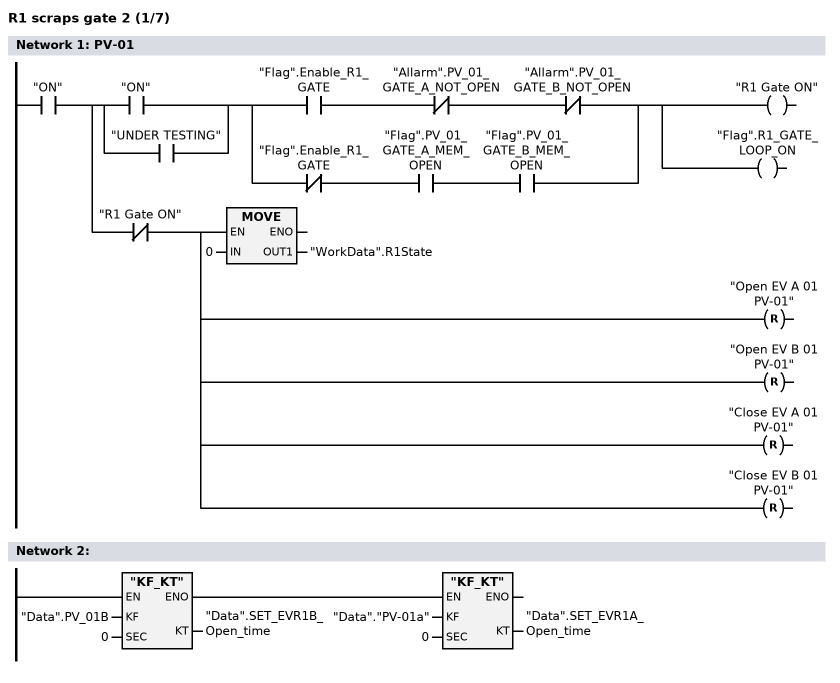
   RUNG wire#powerrail
      Contact( "ON" )
      wire#w1
      Contact( "ON" )
      wire#w2
      Contact( "Flag".Enable_R1_GATE )
      I_Contact( "Allarm".PV_01_GATE_A_NOT_OPEN )
      I_Contact( "Allarm".PV_01_GATE_B_NOT_OPEN )
      wire#w3
      Coil( "R1 Gate ON" )
   END_RUNG
   RUNG wire#w1
      Contact( "UNDER TESTING" )
   END_RUNG wire#w2
   RUNG wire#w2
      I_Contact( "Flag".Enable_R1_GATE )
      Contact( "Flag".PV_01_GATE_A_MEM_OPEN )
      Contact( "Flag".PV_01_GATE_B_MEM_OPEN )
   END_RUNG wire#w3
   RUNG wire#w3
      Coil( "Flag".R1_GATE_LOOP_ON )
   END_RUNG
   RUNG wire#w1
      I_Contact( "R1 Gate ON" )
      wire#w4
      { S7_GenerateENO := "TRUE" } Move(in := 0, out1 => "WorkData".R1State)
   END_RUNG
   RUNG wire#w4
      R_Coil( "Open EV A 01  PV-01" )
   END_RUNG
   RUNG wire#w4
      R_Coil( "Open EV B 01  PV-01" )
   END_RUNG
   RUNG wire#w4
      R_Coil( "Close EV A 01  PV-01" )
   END_RUNG
   RUNG wire#w4
      R_Coil( "Close EV B 01  PV-01" )
   END_RUNG
   // the same network as SCL:
   "R1 Gate ON" := "ON" AND ("ON" OR "UNDER TESTING") AND (("Flag".Enable_R1_GATE AND NOT "Allarm".PV_01_GATE_A_NOT_OPEN AND NOT "Allarm".PV_01_GATE_B_NOT_OPEN) OR (NOT "Flag".Enable_R1_GATE AND "Flag".PV_01_GATE_A_MEM_OPEN AND "Flag".PV_01_GATE_B_MEM_OPEN));
   "Flag".R1_GATE_LOOP_ON := "R1 Gate ON";
   IF "ON" AND NOT "R1 Gate ON" THEN
       "WorkData".R1State := 0;
       "Open EV A 01  PV-01" := FALSE;
       "Open EV B 01  PV-01" := FALSE;
       "Close EV A 01  PV-01" := FALSE;
       "Close EV B 01  PV-01" := FALSE;
   END_IF;
END_REGION

REGION Network 2
   RUNG wire#powerrail
      "KF_KT"(KF := "Data".PV_01B, SEC := 0, KT => "Data".SET_EVR1B_Open_time)
      "KF_KT"(KF := "Data"."PV-01a", SEC := 0, KT => "Data".SET_EVR1A_Open_time)
   END_RUNG
   // the same network as SCL:
   "KF_KT"(KF := "Data".PV_01B, SEC := 0, KT => "Data".SET_EVR1B_Open_time, ENO => #_w1);
   IF #_w1 THEN "KF_KT"(KF := "Data"."PV-01a", SEC := 0, KT => "Data".SET_EVR1A_Open_time); END_IF;
END_REGION

REGION Network 3: R1 gate loop PV-01
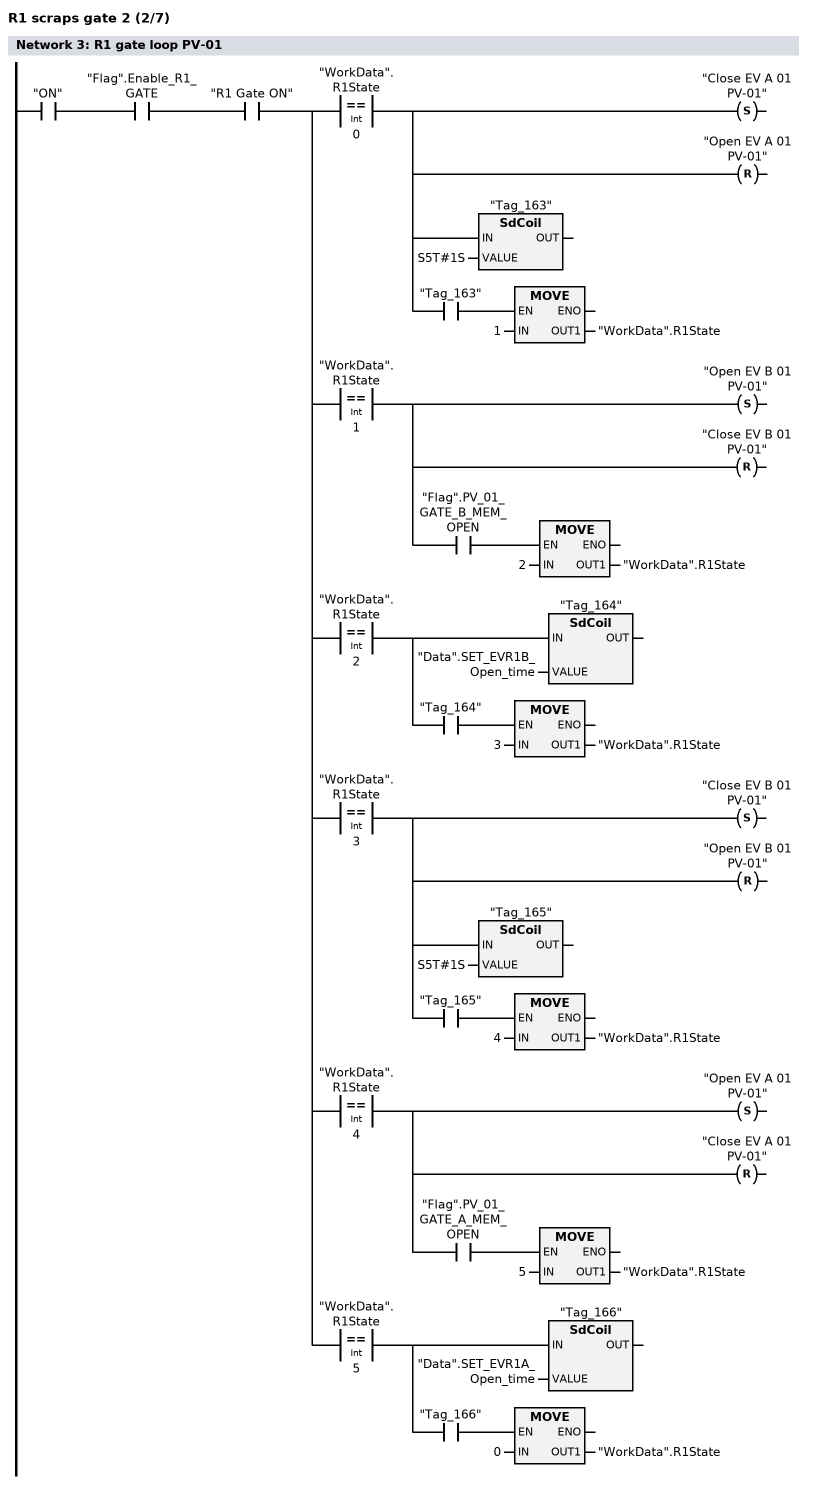
   // no SCL statement known for SdCoil: written as a call
   #_w1 := "ON" AND "Flag".Enable_R1_GATE AND "R1 Gate ON";
   #_w2 := #_w1 AND ("WorkData".R1State = 0);
   IF #_w2 THEN
       "Close EV A 01  PV-01" := TRUE;
       "Open EV A 01  PV-01" := FALSE;
   END_IF;
   SdCoil(in := #_w2, value := S5T#1S, operand := "Tag_163");
   IF #_w2 AND "Tag_163" THEN "WorkData".R1State := 1; END_IF;
   #_w3 := #_w1 AND ("WorkData".R1State = 1);
   IF #_w3 THEN
       "Open EV B 01  PV-01" := TRUE;
       "Close EV B 01  PV-01" := FALSE;
   END_IF;
   IF #_w3 AND "Flag".PV_01_GATE_B_MEM_OPEN THEN "WorkData".R1State := 2; END_IF;
   #_w4 := #_w1 AND ("WorkData".R1State = 2);
   SdCoil(in := #_w4, value := "Data".SET_EVR1B_Open_time, operand := "Tag_164");
   IF #_w4 AND "Tag_164" THEN "WorkData".R1State := 3; END_IF;
   #_w5 := #_w1 AND ("WorkData".R1State = 3);
   IF #_w5 THEN
       "Close EV B 01  PV-01" := TRUE;
       "Open EV B 01  PV-01" := FALSE;
   END_IF;
   SdCoil(in := #_w5, value := S5T#1S, operand := "Tag_165");
   IF #_w5 AND "Tag_165" THEN "WorkData".R1State := 4; END_IF;
   #_w6 := #_w1 AND ("WorkData".R1State = 4);
   IF #_w6 THEN
       "Open EV A 01  PV-01" := TRUE;
       "Close EV A 01  PV-01" := FALSE;
   END_IF;
   IF #_w6 AND "Flag".PV_01_GATE_A_MEM_OPEN THEN "WorkData".R1State := 5; END_IF;
   #_w7 := #_w1 AND ("WorkData".R1State = 5);
   SdCoil(in := #_w7, value := "Data".SET_EVR1A_Open_time, operand := "Tag_166");
   IF #_w7 AND "Tag_166" THEN "WorkData".R1State := 0; END_IF;
END_REGION

REGION Network 4: EVR4 scraps discharge door and Gates selector PV-01
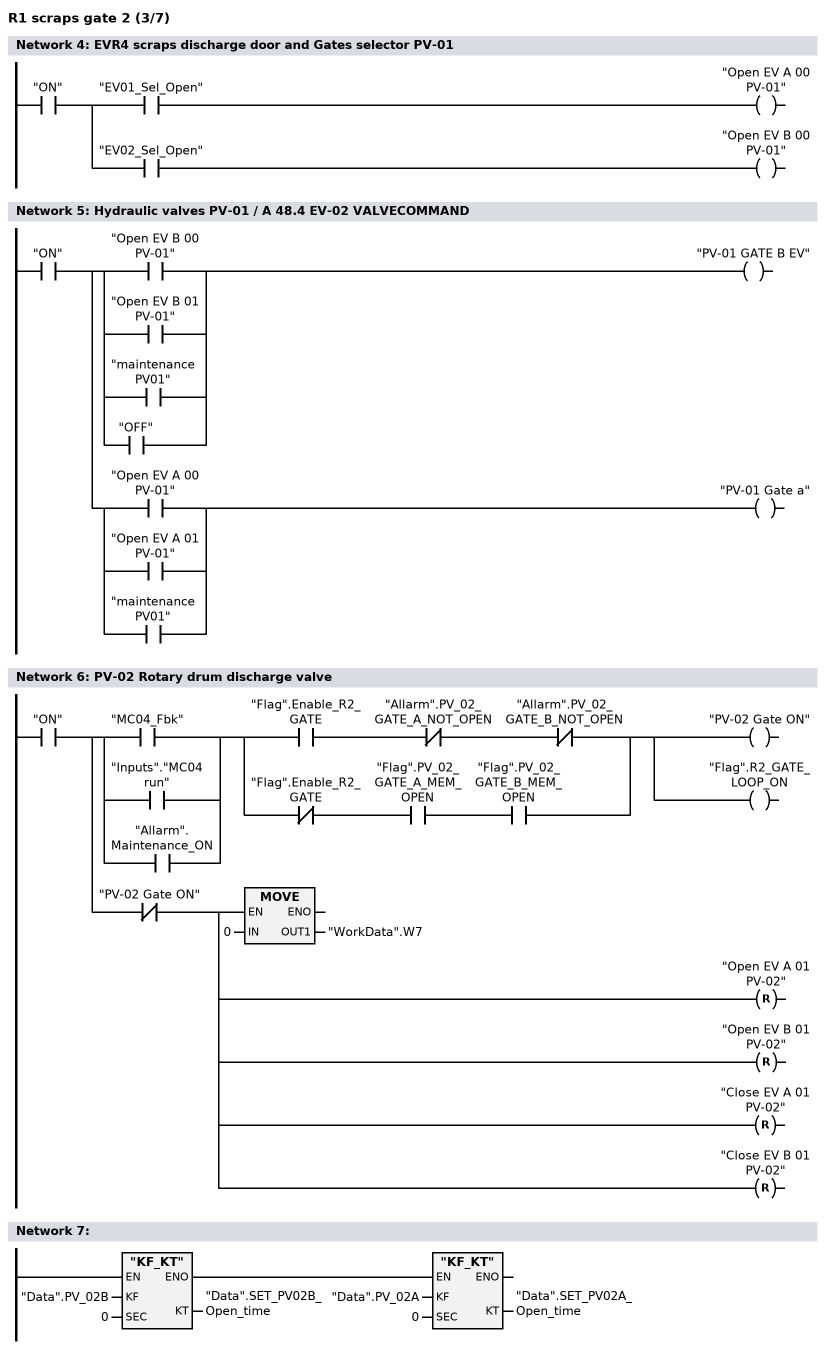
   RUNG wire#powerrail
      Contact( "ON" )
      wire#w1
      Contact( "EV01_Sel_Open" )
      Coil( "Open EV A 00 PV-01" )
   END_RUNG
   RUNG wire#w1
      Contact( "EV02_Sel_Open" )
      Coil( "Open EV B 00  PV-01" )
   END_RUNG
   // the same network as SCL:
   "Open EV A 00 PV-01" := "ON" AND "EV01_Sel_Open";
   "Open EV B 00  PV-01" := "ON" AND "EV02_Sel_Open";
END_REGION

REGION Network 5: Hydraulic valves PV-01 / A 48.4 EV-02 VALVECOMMAND
   RUNG wire#powerrail
      Contact( "ON" )
      wire#w1
      Contact( "Open EV B 00  PV-01" )
      wire#w2
      Coil( "PV-01 GATE B EV" )
   END_RUNG
   RUNG wire#w1
      Contact( "Open EV B 01  PV-01" )
   END_RUNG wire#w2
   RUNG wire#w1
      Contact( "maintenance PV01" )
   END_RUNG wire#w2
   RUNG wire#w1
      Contact( "OFF" )
   END_RUNG wire#w2
   RUNG wire#w1
      Contact( "Open EV A 00 PV-01" )
      wire#w3
      Coil( "PV-01 Gate a" )
   END_RUNG
   RUNG wire#w1
      Contact( "Open EV A 01  PV-01" )
   END_RUNG wire#w3
   RUNG wire#w1
      Contact( "maintenance PV01" )
   END_RUNG wire#w3
   // the same network as SCL:
   "PV-01 GATE B EV" := "ON" AND ("Open EV B 00  PV-01" OR "Open EV B 01  PV-01" OR "maintenance PV01" OR "OFF");
   "PV-01 Gate a" := "ON" AND ("Open EV A 00 PV-01" OR "Open EV A 01  PV-01" OR "maintenance PV01");
END_REGION

REGION Network 6: PV-02 Rotary drum discharge valve
   RUNG wire#powerrail
      Contact( "ON" )
      wire#w1
      Contact( "MC04_Fbk" )
      wire#w2
      Contact( "Flag".Enable_R2_GATE )
      I_Contact( "Allarm".PV_02_GATE_A_NOT_OPEN )
      I_Contact( "Allarm".PV_02_GATE_B_NOT_OPEN )
      wire#w3
      Coil( "PV-02 Gate ON" )
   END_RUNG
   RUNG wire#w1
      Contact( "Inputs"."MC04 run" )
   END_RUNG wire#w2
   RUNG wire#w1
      Contact( "Allarm".Maintenance_ON )
   END_RUNG wire#w2
   RUNG wire#w2
      I_Contact( "Flag".Enable_R2_GATE )
      Contact( "Flag".PV_02_GATE_A_MEM_OPEN )
      Contact( "Flag".PV_02_GATE_B_MEM_OPEN )
   END_RUNG wire#w3
   RUNG wire#w3
      Coil( "Flag".R2_GATE_LOOP_ON )
   END_RUNG
   RUNG wire#w1
      I_Contact( "PV-02 Gate ON" )
      wire#w4
      { S7_GenerateENO := "TRUE" } Move(in := 0, out1 => "WorkData".W7)
   END_RUNG
   RUNG wire#w4
      R_Coil( "Open EV A 01  PV-02" )
   END_RUNG
   RUNG wire#w4
      R_Coil( "Open EV B 01  PV-02" )
   END_RUNG
   RUNG wire#w4
      R_Coil( "Close EV A 01  PV-02" )
   END_RUNG
   RUNG wire#w4
      R_Coil( "Close EV B 01  PV-02" )
   END_RUNG
   // the same network as SCL:
   "PV-02 Gate ON" := "ON" AND ("MC04_Fbk" OR "Inputs"."MC04 run" OR "Allarm".Maintenance_ON) AND (("Flag".Enable_R2_GATE AND NOT "Allarm".PV_02_GATE_A_NOT_OPEN AND NOT "Allarm".PV_02_GATE_B_NOT_OPEN) OR (NOT "Flag".Enable_R2_GATE AND "Flag".PV_02_GATE_A_MEM_OPEN AND "Flag".PV_02_GATE_B_MEM_OPEN));
   "Flag".R2_GATE_LOOP_ON := "PV-02 Gate ON";
   IF "ON" AND NOT "PV-02 Gate ON" THEN
       "WorkData".W7 := 0;
       "Open EV A 01  PV-02" := FALSE;
       "Open EV B 01  PV-02" := FALSE;
       "Close EV A 01  PV-02" := FALSE;
       "Close EV B 01  PV-02" := FALSE;
   END_IF;
END_REGION

REGION Network 7
   RUNG wire#powerrail
      "KF_KT"(KF := "Data".PV_02B, SEC := 0, KT => "Data".SET_PV02B_Open_time)
      "KF_KT"(KF := "Data".PV_02A, SEC := 0, KT => "Data".SET_PV02A_Open_time)
   END_RUNG
   // the same network as SCL:
   "KF_KT"(KF := "Data".PV_02B, SEC := 0, KT => "Data".SET_PV02B_Open_time, ENO => #_w1);
   IF #_w1 THEN "KF_KT"(KF := "Data".PV_02A, SEC := 0, KT => "Data".SET_PV02A_Open_time); END_IF;
END_REGION

REGION Network 8: R1 gate loop PV-02
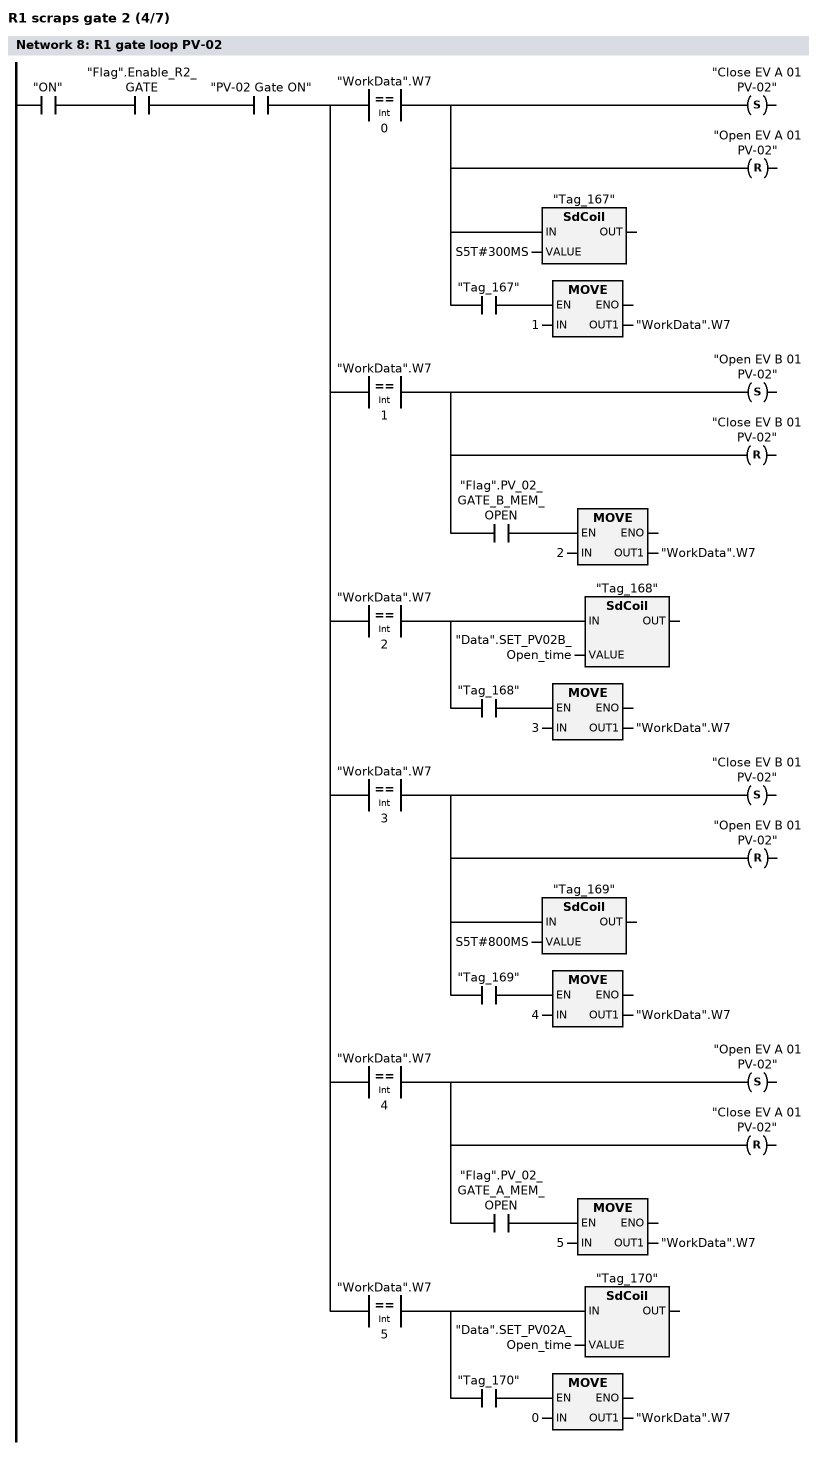
   // no SCL statement known for SdCoil: written as a call
   #_w1 := "ON" AND "Flag".Enable_R2_GATE AND "PV-02 Gate ON";
   #_w2 := #_w1 AND ("WorkData".W7 = 0);
   IF #_w2 THEN
       "Close EV A 01  PV-02" := TRUE;
       "Open EV A 01  PV-02" := FALSE;
   END_IF;
   SdCoil(in := #_w2, value := S5T#300MS, operand := "Tag_167");
   IF #_w2 AND "Tag_167" THEN "WorkData".W7 := 1; END_IF;
   #_w3 := #_w1 AND ("WorkData".W7 = 1);
   IF #_w3 THEN
       "Open EV B 01  PV-02" := TRUE;
       "Close EV B 01  PV-02" := FALSE;
   END_IF;
   IF #_w3 AND "Flag".PV_02_GATE_B_MEM_OPEN THEN "WorkData".W7 := 2; END_IF;
   #_w4 := #_w1 AND ("WorkData".W7 = 2);
   SdCoil(in := #_w4, value := "Data".SET_PV02B_Open_time, operand := "Tag_168");
   IF #_w4 AND "Tag_168" THEN "WorkData".W7 := 3; END_IF;
   #_w5 := #_w1 AND ("WorkData".W7 = 3);
   IF #_w5 THEN
       "Close EV B 01  PV-02" := TRUE;
       "Open EV B 01  PV-02" := FALSE;
   END_IF;
   SdCoil(in := #_w5, value := S5T#800MS, operand := "Tag_169");
   IF #_w5 AND "Tag_169" THEN "WorkData".W7 := 4; END_IF;
   #_w6 := #_w1 AND ("WorkData".W7 = 4);
   IF #_w6 THEN
       "Open EV A 01  PV-02" := TRUE;
       "Close EV A 01  PV-02" := FALSE;
   END_IF;
   IF #_w6 AND "Flag".PV_02_GATE_A_MEM_OPEN THEN "WorkData".W7 := 5; END_IF;
   #_w7 := #_w1 AND ("WorkData".W7 = 5);
   SdCoil(in := #_w7, value := "Data".SET_PV02A_Open_time, operand := "Tag_170");
   IF #_w7 AND "Tag_170" THEN "WorkData".W7 := 0; END_IF;
END_REGION

REGION Network 9: EVR4 scraps discharge door and Gates selector PV-02
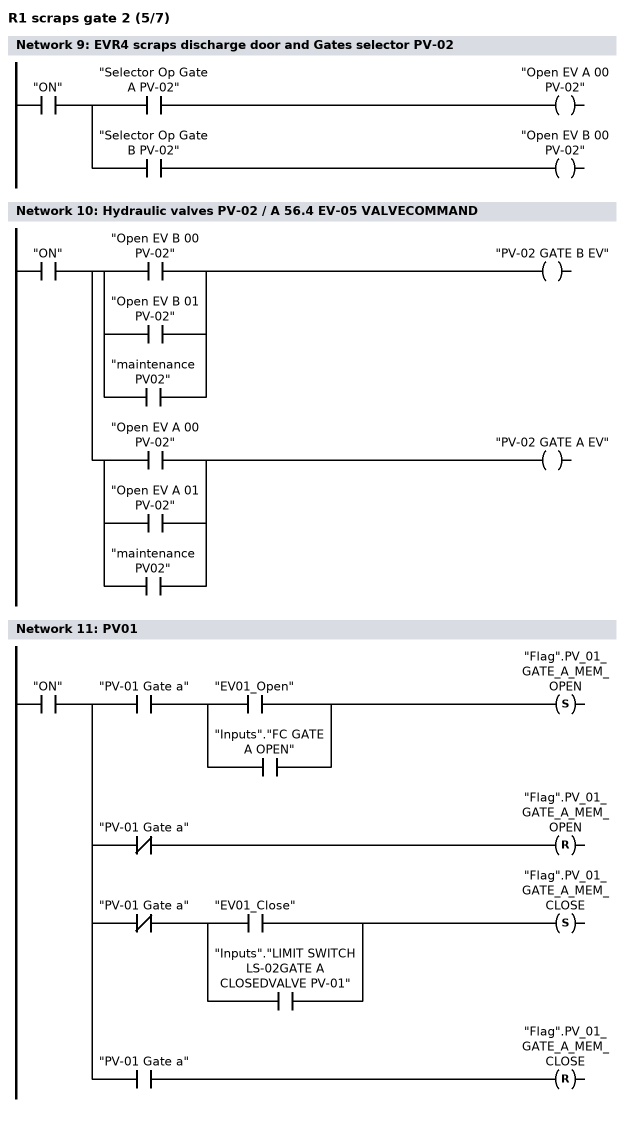
   RUNG wire#powerrail
      Contact( "ON" )
      wire#w1
      Contact( "Selector Op Gate A PV-02" )
      Coil( "Open EV A 00 PV-02" )
   END_RUNG
   RUNG wire#w1
      Contact( "Selector Op Gate B PV-02" )
      Coil( "Open EV B 00  PV-02" )
   END_RUNG
   // the same network as SCL:
   "Open EV A 00 PV-02" := "ON" AND "Selector Op Gate A PV-02";
   "Open EV B 00  PV-02" := "ON" AND "Selector Op Gate B PV-02";
END_REGION

REGION Network 10: Hydraulic valves PV-02 / A 56.4 EV-05 VALVECOMMAND
   RUNG wire#powerrail
      Contact( "ON" )
      wire#w1
      Contact( "Open EV B 00  PV-02" )
      wire#w2
      Coil( "PV-02 GATE B EV" )
   END_RUNG
   RUNG wire#w1
      Contact( "Open EV B 01  PV-02" )
   END_RUNG wire#w2
   RUNG wire#w1
      Contact( "maintenance PV02" )
   END_RUNG wire#w2
   RUNG wire#w1
      Contact( "Open EV A 00 PV-02" )
      wire#w3
      Coil( "PV-02 GATE A EV" )
   END_RUNG
   RUNG wire#w1
      Contact( "Open EV A 01  PV-02" )
   END_RUNG wire#w3
   RUNG wire#w1
      Contact( "maintenance PV02" )
   END_RUNG wire#w3
   // the same network as SCL:
   "PV-02 GATE B EV" := "ON" AND ("Open EV B 00  PV-02" OR "Open EV B 01  PV-02" OR "maintenance PV02");
   "PV-02 GATE A EV" := "ON" AND ("Open EV A 00 PV-02" OR "Open EV A 01  PV-02" OR "maintenance PV02");
END_REGION

REGION Network 11: PV01
   RUNG wire#powerrail
      Contact( "ON" )
      wire#w1
      Contact( "PV-01 Gate a" )
      wire#w2
      Contact( "EV01_Open" )
      wire#w3
      S_Coil( "Flag".PV_01_GATE_A_MEM_OPEN )
   END_RUNG
   RUNG wire#w2
      Contact( "Inputs"."FC GATE A OPEN" )
   END_RUNG wire#w3
   RUNG wire#w1
      I_Contact( "PV-01 Gate a" )
      R_Coil( "Flag".PV_01_GATE_A_MEM_OPEN )
   END_RUNG
   RUNG wire#w1
      I_Contact( "PV-01 Gate a" )
      wire#w4
      Contact( "EV01_Close" )
      wire#w5
      S_Coil( "Flag".PV_01_GATE_A_MEM_CLOSE )
   END_RUNG
   RUNG wire#w4
      Contact( "Inputs"."LIMIT SWITCH LS-02GATE A CLOSEDVALVE PV-01" )
   END_RUNG wire#w5
   RUNG wire#w1
      Contact( "PV-01 Gate a" )
      R_Coil( "Flag".PV_01_GATE_A_MEM_CLOSE )
   END_RUNG
   // the same network as SCL:
   IF "ON" AND "PV-01 Gate a" AND ("EV01_Open" OR "Inputs"."FC GATE A OPEN") THEN
       "Flag".PV_01_GATE_A_MEM_OPEN := TRUE;
   END_IF;
   IF "ON" AND NOT "PV-01 Gate a" THEN "Flag".PV_01_GATE_A_MEM_OPEN := FALSE; END_IF;
   IF "ON" AND NOT "PV-01 Gate a" AND ("EV01_Close" OR "Inputs"."LIMIT SWITCH LS-02GATE A CLOSEDVALVE PV-01") THEN
       "Flag".PV_01_GATE_A_MEM_CLOSE := TRUE;
   END_IF;
   IF "ON" AND "PV-01 Gate a" THEN "Flag".PV_01_GATE_A_MEM_CLOSE := FALSE; END_IF;
END_REGION

REGION Network 12: PV01
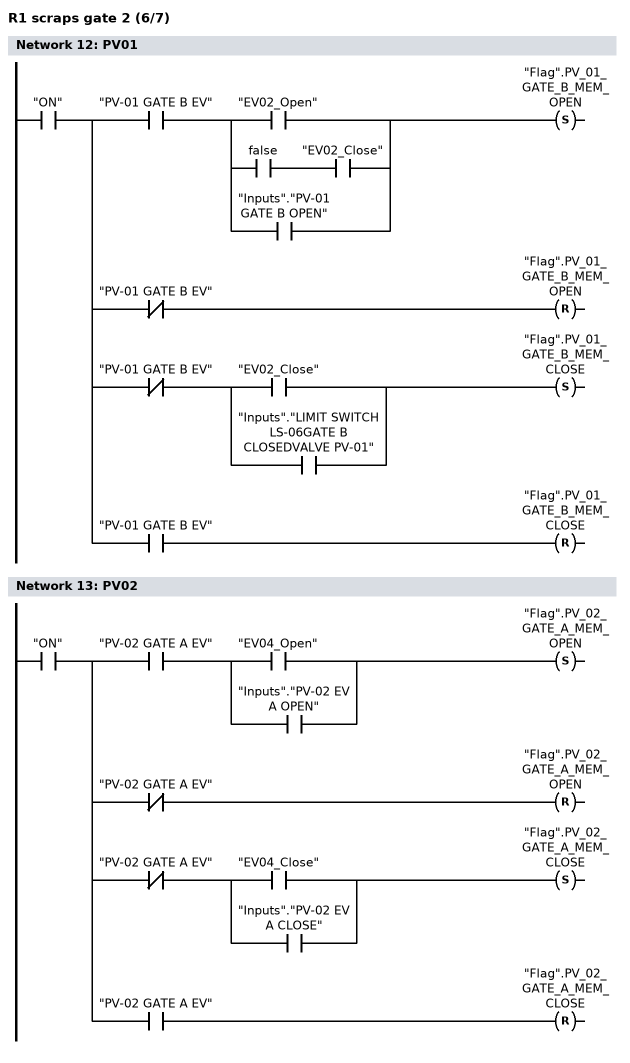
   RUNG wire#powerrail
      Contact( "ON" )
      wire#w1
      Contact( "PV-01 GATE B EV" )
      wire#w2
      Contact( "EV02_Open" )
      wire#w3
      S_Coil( "Flag".PV_01_GATE_B_MEM_OPEN )
   END_RUNG
   RUNG wire#w2
      Contact( false )
      Contact( "EV02_Close" )
   END_RUNG wire#w3
   RUNG wire#w2
      Contact( "Inputs"."PV-01 GATE B OPEN" )
   END_RUNG wire#w3
   RUNG wire#w1
      I_Contact( "PV-01 GATE B EV" )
      R_Coil( "Flag".PV_01_GATE_B_MEM_OPEN )
   END_RUNG
   RUNG wire#w1
      I_Contact( "PV-01 GATE B EV" )
      wire#w4
      Contact( "EV02_Close" )
      wire#w5
      S_Coil( "Flag".PV_01_GATE_B_MEM_CLOSE )
   END_RUNG
   RUNG wire#w4
      Contact( "Inputs"."LIMIT SWITCH LS-06GATE B CLOSEDVALVE PV-01" )
   END_RUNG wire#w5
   RUNG wire#w1
      Contact( "PV-01 GATE B EV" )
      R_Coil( "Flag".PV_01_GATE_B_MEM_CLOSE )
   END_RUNG
   // the same network as SCL:
   IF "ON" AND "PV-01 GATE B EV" AND ("EV02_Open" OR (false AND "EV02_Close") OR "Inputs"."PV-01 GATE B OPEN") THEN
       "Flag".PV_01_GATE_B_MEM_OPEN := TRUE;
   END_IF;
   IF "ON" AND NOT "PV-01 GATE B EV" THEN "Flag".PV_01_GATE_B_MEM_OPEN := FALSE; END_IF;
   IF "ON" AND NOT "PV-01 GATE B EV" AND ("EV02_Close" OR "Inputs"."LIMIT SWITCH LS-06GATE B CLOSEDVALVE PV-01") THEN
       "Flag".PV_01_GATE_B_MEM_CLOSE := TRUE;
   END_IF;
   IF "ON" AND "PV-01 GATE B EV" THEN "Flag".PV_01_GATE_B_MEM_CLOSE := FALSE; END_IF;
END_REGION

REGION Network 13: PV02
   RUNG wire#powerrail
      Contact( "ON" )
      wire#w1
      Contact( "PV-02 GATE A EV" )
      wire#w2
      Contact( "EV04_Open" )
      wire#w3
      S_Coil( "Flag".PV_02_GATE_A_MEM_OPEN )
   END_RUNG
   RUNG wire#w2
      Contact( "Inputs"."PV-02 EV A OPEN" )
   END_RUNG wire#w3
   RUNG wire#w1
      I_Contact( "PV-02 GATE A EV" )
      R_Coil( "Flag".PV_02_GATE_A_MEM_OPEN )
   END_RUNG
   RUNG wire#w1
      I_Contact( "PV-02 GATE A EV" )
      wire#w4
      Contact( "EV04_Close" )
      wire#w5
      S_Coil( "Flag".PV_02_GATE_A_MEM_CLOSE )
   END_RUNG
   RUNG wire#w4
      Contact( "Inputs"."PV-02 EV A CLOSE" )
   END_RUNG wire#w5
   RUNG wire#w1
      Contact( "PV-02 GATE A EV" )
      R_Coil( "Flag".PV_02_GATE_A_MEM_CLOSE )
   END_RUNG
   // the same network as SCL:
   IF "ON" AND "PV-02 GATE A EV" AND ("EV04_Open" OR "Inputs"."PV-02 EV A OPEN") THEN
       "Flag".PV_02_GATE_A_MEM_OPEN := TRUE;
   END_IF;
   IF "ON" AND NOT "PV-02 GATE A EV" THEN "Flag".PV_02_GATE_A_MEM_OPEN := FALSE; END_IF;
   IF "ON" AND NOT "PV-02 GATE A EV" AND ("EV04_Close" OR "Inputs"."PV-02 EV A CLOSE") THEN
       "Flag".PV_02_GATE_A_MEM_CLOSE := TRUE;
   END_IF;
   IF "ON" AND "PV-02 GATE A EV" THEN "Flag".PV_02_GATE_A_MEM_CLOSE := FALSE; END_IF;
END_REGION

REGION Network 14: PV02
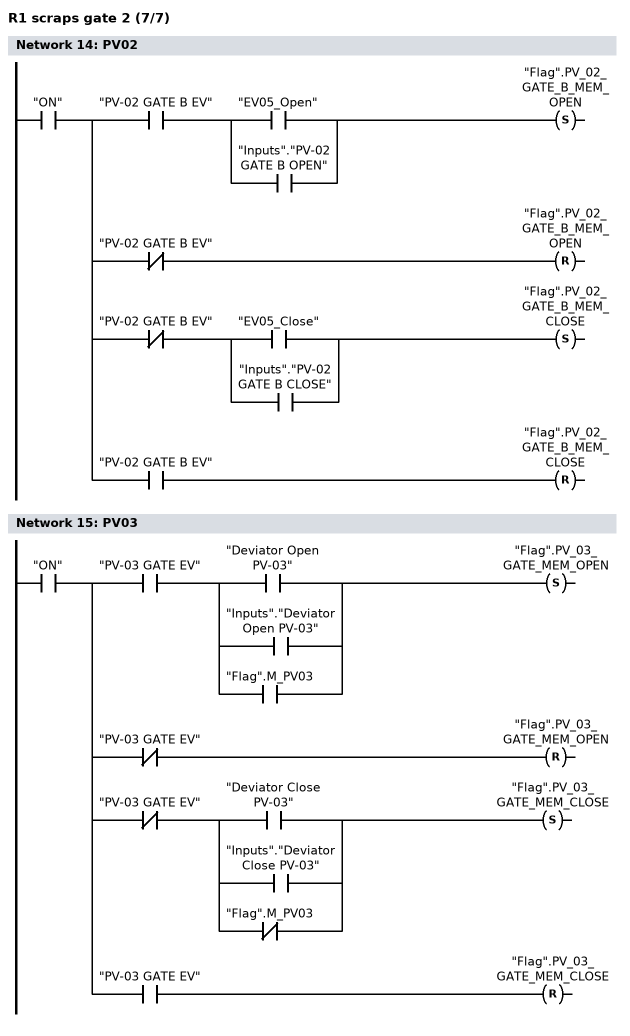
   RUNG wire#powerrail
      Contact( "ON" )
      wire#w1
      Contact( "PV-02 GATE B EV" )
      wire#w2
      Contact( "EV05_Open" )
      wire#w3
      S_Coil( "Flag".PV_02_GATE_B_MEM_OPEN )
   END_RUNG
   RUNG wire#w2
      Contact( "Inputs"."PV-02 GATE B OPEN" )
   END_RUNG wire#w3
   RUNG wire#w1
      I_Contact( "PV-02 GATE B EV" )
      R_Coil( "Flag".PV_02_GATE_B_MEM_OPEN )
   END_RUNG
   RUNG wire#w1
      I_Contact( "PV-02 GATE B EV" )
      wire#w4
      Contact( "EV05_Close" )
      wire#w5
      S_Coil( "Flag".PV_02_GATE_B_MEM_CLOSE )
   END_RUNG
   RUNG wire#w4
      Contact( "Inputs"."PV-02 GATE B CLOSE" )
   END_RUNG wire#w5
   RUNG wire#w1
      Contact( "PV-02 GATE B EV" )
      R_Coil( "Flag".PV_02_GATE_B_MEM_CLOSE )
   END_RUNG
   // the same network as SCL:
   IF "ON" AND "PV-02 GATE B EV" AND ("EV05_Open" OR "Inputs"."PV-02 GATE B OPEN") THEN
       "Flag".PV_02_GATE_B_MEM_OPEN := TRUE;
   END_IF;
   IF "ON" AND NOT "PV-02 GATE B EV" THEN "Flag".PV_02_GATE_B_MEM_OPEN := FALSE; END_IF;
   IF "ON" AND NOT "PV-02 GATE B EV" AND ("EV05_Close" OR "Inputs"."PV-02 GATE B CLOSE") THEN
       "Flag".PV_02_GATE_B_MEM_CLOSE := TRUE;
   END_IF;
   IF "ON" AND "PV-02 GATE B EV" THEN "Flag".PV_02_GATE_B_MEM_CLOSE := FALSE; END_IF;
END_REGION

REGION Network 15: PV03
   RUNG wire#powerrail
      Contact( "ON" )
      wire#w1
      Contact( "PV-03 GATE EV" )
      wire#w2
      Contact( "Deviator Open PV-03" )
      wire#w3
      S_Coil( "Flag".PV_03_GATE_MEM_OPEN )
   END_RUNG
   RUNG wire#w2
      Contact( "Inputs"."Deviator Open PV-03" )
   END_RUNG wire#w3
   RUNG wire#w2
      Contact( "Flag".M_PV03 )
   END_RUNG wire#w3
   RUNG wire#w1
      I_Contact( "PV-03 GATE EV" )
      R_Coil( "Flag".PV_03_GATE_MEM_OPEN )
   END_RUNG
   RUNG wire#w1
      I_Contact( "PV-03 GATE EV" )
      wire#w4
      Contact( "Deviator Close PV-03" )
      wire#w5
      S_Coil( "Flag".PV_03_GATE_MEM_CLOSE )
   END_RUNG
   RUNG wire#w4
      Contact( "Inputs"."Deviator Close PV-03" )
   END_RUNG wire#w5
   RUNG wire#w4
      I_Contact( "Flag".M_PV03 )
   END_RUNG wire#w5
   RUNG wire#w1
      Contact( "PV-03 GATE EV" )
      R_Coil( "Flag".PV_03_GATE_MEM_CLOSE )
   END_RUNG
   // the same network as SCL:
   IF "ON" AND "PV-03 GATE EV" AND ("Deviator Open PV-03" OR "Inputs"."Deviator Open PV-03" OR "Flag".M_PV03) THEN
       "Flag".PV_03_GATE_MEM_OPEN := TRUE;
   END_IF;
   IF "ON" AND NOT "PV-03 GATE EV" THEN "Flag".PV_03_GATE_MEM_OPEN := FALSE; END_IF;
   IF "ON" AND NOT "PV-03 GATE EV" AND ("Deviator Close PV-03" OR "Inputs"."Deviator Close PV-03" OR NOT "Flag".M_PV03) THEN
       "Flag".PV_03_GATE_MEM_CLOSE := TRUE;
   END_IF;
   IF "ON" AND "PV-03 GATE EV" THEN "Flag".PV_03_GATE_MEM_CLOSE := FALSE; END_IF;
END_REGION
END_FUNCTION

FUNCTION "KF_KT" : Void   // FC109, STL
TITLE = Conversione tempo KF => KT - Max. 9990 secondi / Converion time KF=>KT - Max. 9990 seconds
{ S7_Optimized_Access := 'FALSE' }
VERSION : 0.1
   VAR_INPUT
      KF : Int;   // Secondi o decimi / Seconds or tenths
      SEC : Bool;   // TRUE = secondi, FALSE = decimi / TRUE = seconds, FALSE = tenths
   END_VAR
   VAR_OUTPUT
      KT : Word;
   END_VAR
BEGIN

REGION Network 1
   // Converte il valore di tempo KF espresso in secondi o in decimi di secondo nel 
   // corrispondente preset in formato S5T (KT); in SEC occorre specificare TRUE se
   // il valore di partenza è espresso in secondi, FALSE se in decimi.
   // Converts the KF time value expressed in seconds or tenths of a second to 
   // corresponding preset in S5T (KT) format; in SEC you must specify TRUE if
   // the starting value is expressed in seconds, FALSE if in tenths

         L     0;
         T     #KT;
         L     #KF;  // tempo in secondi o decimi
         >=I;
         BEC;  // esci se <= 0

         AN    #SEC;
         JC    X1;  // se secondi
         L     10;  // x 10
         *I;  // Tempo in decimi

   // Tra 0 e 9.9 secondi
   X1:   L     99;
         >D;
         JC    X2;
         TAK;  // Tempo in decimi
         ITB;  // Converti in BCD
         SLW   4;  // aggiungi uno zero a destra (x10)
         JU    ESC;  // Base 0 = decine di ms

   // Tra 10.0 e 99.9 secondi
   X2:   TAK;  // Tempo in decimi
         L     999;
         >D;
         JC    X3;
         TAK;  // Tempo in decimi
         ITB;  // Converti in BCD
         L     16#1000;  // Base 1 = decimi
         JU    OR;

   // Tra 100.0 e 999.9 secondi
   X3:   TAK;  // Tempo in decimi
         +     5;  // +5 per arrotondamento
         L     9999;
         >D;
         JC    X4;
         TAK;  // Tempo in decimi
         DTB;  // converti in BCD
         SRD   4;  // Sposta a destra di 1 cifra (/10)
         L     16#2000;  // Base 2 = secondi
         JU    OR;

   // Tra 1000.0 e 9990.0 secondi
   X4:   TAK;  // Tempo in decimi
         +     45;  // +50 (45+5) per arrotondamento
         L     99900;
         >D;
         JC    X5;
         TAK;  // Tempo in decimi
         DTB;  // converti in BCD
         SRD   8;  // Sposta a destra di 2 cifre (/100)
         L     16#3000;  // Base 3 = decine di secondi
         JU    OR;

   // Oltre 9990.0 secondi
   X5:   L     16#3999;  // Massimo tempo possibile
         JU    ESC;

   // Uscita
   OR:   OW;  // Aggiungi la base
   ESC:  T     #KT;  // Uscita
END_REGION
END_FUNCTION

ORGANIZATION_BLOCK "Main"   // OB1, LAD, ProgramCycle
TITLE = Main program
{ S7_Optimized_Access := 'FALSE' }
VERSION : 0.1
   VAR_TEMP
      TodayDate : Date;
      ReadClkRetValue : Int;
      TodayDateTime : Date_And_Time;
      spare : DWord;
      spare_1 : DWord;
      spare_2 : DWord;
   END_VAR
   VAR_TEMP   // added for the SCL form of the ladder/FBD networks
      _w1 : Bool;
      _w2 : Bool;
      _w3 : Bool;
   END_VAR
BEGIN

REGION Network 1: SIMULATION
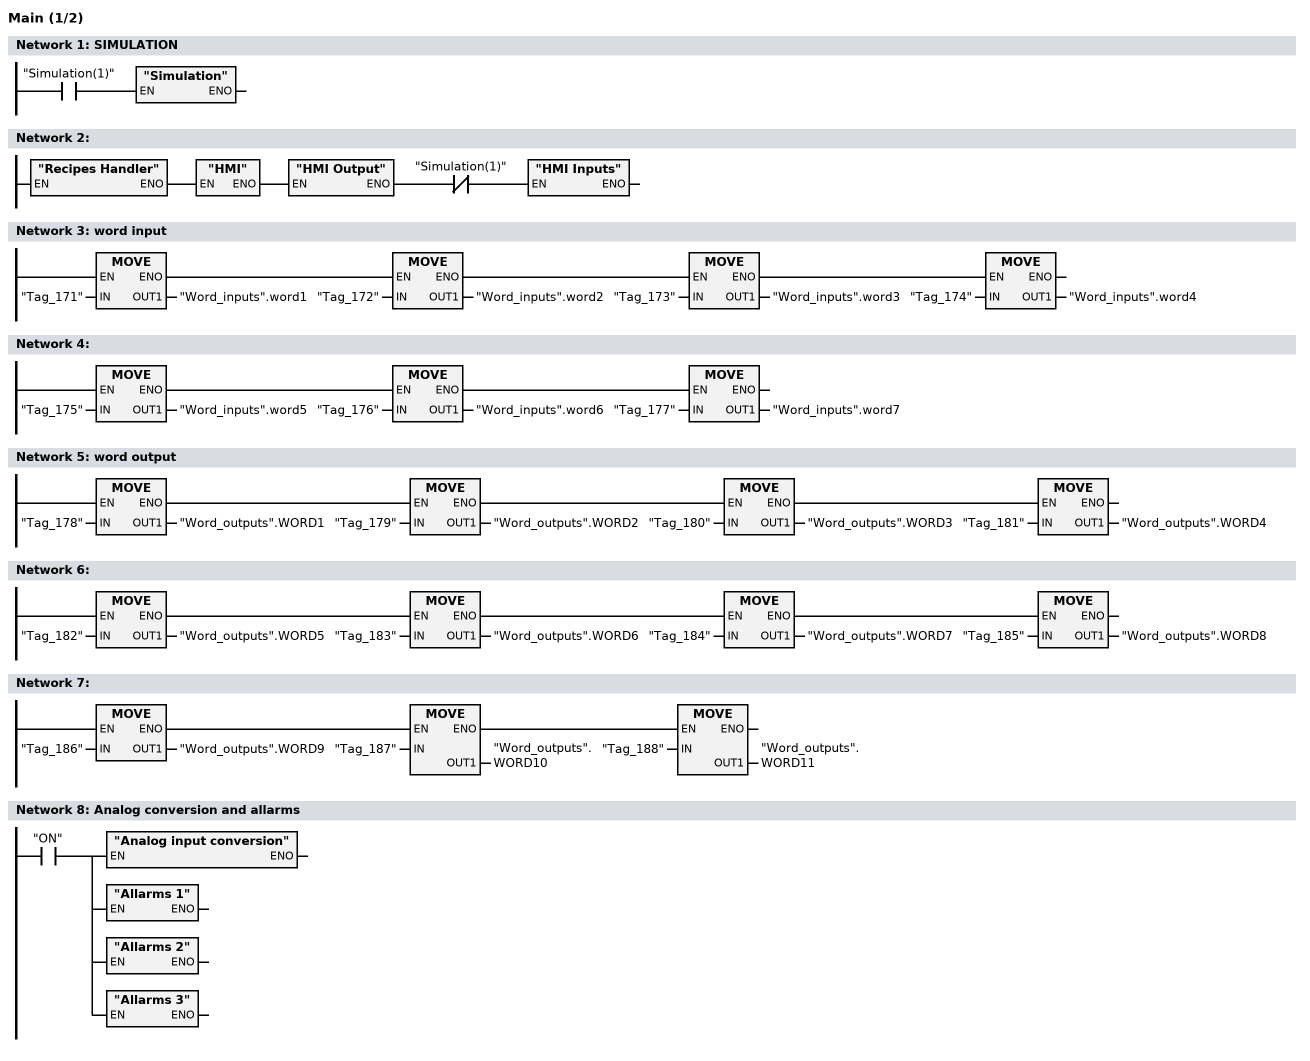
   RUNG wire#powerrail
      Contact( "Simulation(1)" )
      "Simulation"()
   END_RUNG
   // the same network as SCL:
   IF "Simulation(1)" THEN "Simulation"(); END_IF;
END_REGION

REGION Network 2
   RUNG wire#powerrail
      "Recipes Handler"()
      "HMI"()
      "HMI Output"()
      I_Contact( "Simulation(1)" )
      "HMI Inputs"()
   END_RUNG
   // the same network as SCL:
   "Recipes Handler"(ENO => #_w1);
   "HMI"(EN := #_w1, ENO => #_w2);
   "HMI Output"(EN := #_w2, ENO => #_w3);
   IF #_w3 AND NOT "Simulation(1)" THEN "HMI Inputs"(); END_IF;
END_REGION

REGION Network 3: word input
   RUNG wire#powerrail
      { S7_GenerateENO := "TRUE" } Move(in := "Tag_171", out1 => "Word_inputs".word1)
      { S7_GenerateENO := "TRUE" } Move(in := "Tag_172", out1 => "Word_inputs".word2)
      { S7_GenerateENO := "TRUE" } Move(in := "Tag_173", out1 => "Word_inputs".word3)
      { S7_GenerateENO := "TRUE" } Move(in := "Tag_174", out1 => "Word_inputs".word4)
   END_RUNG
   // the same network as SCL:
   // ENO of a box is taken as its EN; it also drops when the box reports an error
   "Word_inputs".word1 := "Tag_171";
   "Word_inputs".word2 := "Tag_172";
   "Word_inputs".word3 := "Tag_173";
   "Word_inputs".word4 := "Tag_174";
END_REGION

REGION Network 4
   RUNG wire#powerrail
      { S7_GenerateENO := "TRUE" } Move(in := "Tag_175", out1 => "Word_inputs".word5)
      { S7_GenerateENO := "TRUE" } Move(in := "Tag_176", out1 => "Word_inputs".word6)
      { S7_GenerateENO := "TRUE" } Move(in := "Tag_177", out1 => "Word_inputs".word7)
   END_RUNG
   // the same network as SCL:
   // ENO of a box is taken as its EN; it also drops when the box reports an error
   "Word_inputs".word5 := "Tag_175";
   "Word_inputs".word6 := "Tag_176";
   "Word_inputs".word7 := "Tag_177";
END_REGION

REGION Network 5: word output
   RUNG wire#powerrail
      { S7_GenerateENO := "TRUE" } Move(in := "Tag_178", out1 => "Word_outputs".WORD1)
      { S7_GenerateENO := "TRUE" } Move(in := "Tag_179", out1 => "Word_outputs".WORD2)
      { S7_GenerateENO := "TRUE" } Move(in := "Tag_180", out1 => "Word_outputs".WORD3)
      { S7_GenerateENO := "TRUE" } Move(in := "Tag_181", out1 => "Word_outputs".WORD4)
   END_RUNG
   // the same network as SCL:
   // ENO of a box is taken as its EN; it also drops when the box reports an error
   "Word_outputs".WORD1 := "Tag_178";
   "Word_outputs".WORD2 := "Tag_179";
   "Word_outputs".WORD3 := "Tag_180";
   "Word_outputs".WORD4 := "Tag_181";
END_REGION

REGION Network 6
   RUNG wire#powerrail
      { S7_GenerateENO := "TRUE" } Move(in := "Tag_182", out1 => "Word_outputs".WORD5)
      { S7_GenerateENO := "TRUE" } Move(in := "Tag_183", out1 => "Word_outputs".WORD6)
      { S7_GenerateENO := "TRUE" } Move(in := "Tag_184", out1 => "Word_outputs".WORD7)
      { S7_GenerateENO := "TRUE" } Move(in := "Tag_185", out1 => "Word_outputs".WORD8)
   END_RUNG
   // the same network as SCL:
   // ENO of a box is taken as its EN; it also drops when the box reports an error
   "Word_outputs".WORD5 := "Tag_182";
   "Word_outputs".WORD6 := "Tag_183";
   "Word_outputs".WORD7 := "Tag_184";
   "Word_outputs".WORD8 := "Tag_185";
END_REGION

REGION Network 7
   RUNG wire#powerrail
      { S7_GenerateENO := "TRUE" } Move(in := "Tag_186", out1 => "Word_outputs".WORD9)
      { S7_GenerateENO := "TRUE" } Move(in := "Tag_187", out1 => "Word_outputs".WORD10)
      { S7_GenerateENO := "TRUE" } Move(in := "Tag_188", out1 => "Word_outputs".WORD11)
   END_RUNG
   // the same network as SCL:
   // ENO of a box is taken as its EN; it also drops when the box reports an error
   "Word_outputs".WORD9 := "Tag_186";
   "Word_outputs".WORD10 := "Tag_187";
   "Word_outputs".WORD11 := "Tag_188";
END_REGION

REGION Network 8: Analog conversion and allarms
   RUNG wire#powerrail
      Contact( "ON" )
      wire#w1
      "Analog input conversion"()
   END_RUNG
   RUNG wire#w1
      "Allarms 1"()
   END_RUNG
   RUNG wire#w1
      "Allarms 2"()
   END_RUNG
   RUNG wire#w1
      "Allarms 3"()
   END_RUNG
   // the same network as SCL:
   #_w1 := "ON";
   IF #_w1 THEN
       "Analog input conversion"();
       "Allarms 1"();
       "Allarms 2"();
       "Allarms 3"();
   END_IF;
END_REGION

REGION Network 9: Motors valve and burner
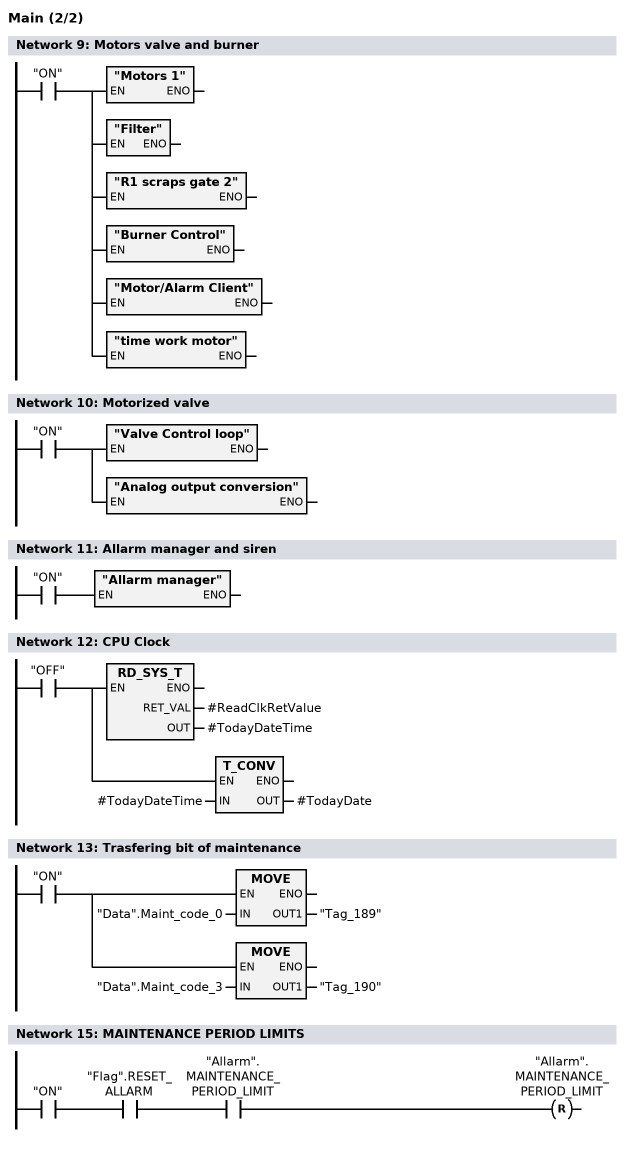
   RUNG wire#powerrail
      Contact( "ON" )
      wire#w1
      "Motors 1"()
   END_RUNG
   RUNG wire#w1
      "Filter"()
   END_RUNG
   RUNG wire#w1
      "R1 scraps gate 2"()
   END_RUNG
   RUNG wire#w1
      "Burner Control"()
   END_RUNG
   RUNG wire#w1
      "Motor/Alarm Client"()
   END_RUNG
   RUNG wire#w1
      "time work motor"()
   END_RUNG
   // the same network as SCL:
   #_w1 := "ON";
   IF #_w1 THEN
       "Motors 1"();
       "Filter"();
       "R1 scraps gate 2"();
       "Burner Control"();
       "Motor/Alarm Client"();
       "time work motor"();
   END_IF;
END_REGION

REGION Network 10: Motorized valve
   RUNG wire#powerrail
      Contact( "ON" )
      wire#w1
      "Valve Control loop"()
   END_RUNG
   RUNG wire#w1
      "Analog output conversion"()
   END_RUNG
   // the same network as SCL:
   #_w1 := "ON";
   IF #_w1 THEN
       "Valve Control loop"();
       "Analog output conversion"();
   END_IF;
END_REGION

REGION Network 11: Allarm manager and siren
   RUNG wire#powerrail
      Contact( "ON" )
      "Allarm manager"()
   END_RUNG
   // the same network as SCL:
   IF "ON" THEN "Allarm manager"(); END_IF;
END_REGION

REGION Network 12: CPU Clock
   #_w1 := "OFF";
   IF #_w1 THEN
       #ReadClkRetValue := RD_SYS_T(OUT => #TodayDateTime);
       #TodayDate := T_CONV(IN := #TodayDateTime);
   END_IF;
END_REGION

REGION Network 13: Trasfering bit of maintenance
   RUNG wire#powerrail
      Contact( "ON" )
      wire#w1
      { S7_GenerateENO := "TRUE" } Move(in := "Data".Maint_code_0, out1 => "Tag_189")
   END_RUNG
   RUNG wire#w1
      { S7_GenerateENO := "TRUE" } Move(in := "Data".Maint_code_3, out1 => "Tag_190")
   END_RUNG
   // the same network as SCL:
   IF "ON" THEN
       "Tag_189" := "Data".Maint_code_0;
       "Tag_190" := "Data".Maint_code_3;
   END_IF;
END_REGION

REGION Network 14 (STL): MAINTENANCE PERIOD LIMITS
         L     "Data".Maint_code_1;

         L     16972;
         ==I;
         JC    M001;

         CALL  RD_SYS_T
         ( RET_VAL := #ReadClkRetValue,
           OUT     := #TodayDateTime
         );

         CALL  T_CONV
         ( IN  := #TodayDateTime,
           OUT := #TodayDate
         );

         L     #TodayDate;
         L     D#2026-01-01;


         >=I;
         S     "Allarm".MAINTENANCE_PERIOD_LIMIT;

   M001: NOP   0;
END_REGION

REGION Network 15: MAINTENANCE PERIOD LIMITS
   RUNG wire#powerrail
      Contact( "ON" )
      Contact( "Flag".RESET_ALLARM )
      Contact( "Allarm".MAINTENANCE_PERIOD_LIMIT )
      R_Coil( "Allarm".MAINTENANCE_PERIOD_LIMIT )
   END_RUNG
   // the same network as SCL:
   IF "ON" AND "Flag".RESET_ALLARM AND "Allarm".MAINTENANCE_PERIOD_LIMIT THEN
       "Allarm".MAINTENANCE_PERIOD_LIMIT := FALSE;
   END_IF;
END_REGION
END_ORGANIZATION_BLOCK

ORGANIZATION_BLOCK "TOD_INT0"   // OB10, LAD, TimeOfDay
TITLE = "Time of Day Interrupt"
{ S7_Optimized_Access := 'FALSE' }
VERSION : 0.1
   VAR_TEMP
      OB10_EV_CLASS : Byte;   // Bits 0-3 = 1 (Coming event), Bits 4-7 = 1 (Event class 1)
      OB10_STRT_INFO : Byte;   // 16#11 (OB 10 has started)
      OB10_PRIORITY : Byte;   // Priority of OB Execution
      OB10_OB_NUMBR : Byte;   // 10 (Organization block 10, OB10)
      OB10_RESERVED_1 : Byte;   // Reserved for system
      OB10_RESERVED_2 : Byte;   // Reserved for system
      OB10_PERIOD_EXE : Word;   // Period of execution (once, per minute/hour/day/week/month/year)
      OB10_RESERVED_3 : Int;   // Reserved for system
      OB10_RESERVED_4 : Int;   // Reserved for system
      OB10_DATE_TIME : Date_And_Time;   // Date and time OB10 started
   END_VAR
BEGIN

REGION Network 1
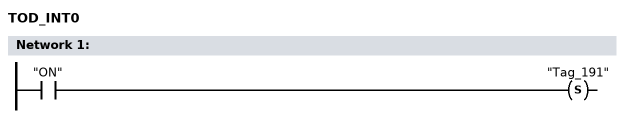
   RUNG wire#powerrail
      Contact( "ON" )
      S_Coil( "Tag_191" )
   END_RUNG
   // the same network as SCL:
   IF "ON" THEN "Tag_191" := TRUE; END_IF;
END_REGION
END_ORGANIZATION_BLOCK

ORGANIZATION_BLOCK "CYC_INT2 Ogni 1s"   // OB32, LAD, CyclicInterrupt
TITLE = "Cyclic Interrupt 1 second"
{ S7_Optimized_Access := 'FALSE' }
VERSION : 0.1
   VAR_TEMP
      Manuale : Bool;
      SPValue : Real;
      ProcValue : Real;
      ManValue : Real;
      OutValue : Real;
      MaxValue : Real;
      TestP : Real;
      TestI : Real;
      TestD : Real;
      FFWD : Real;
      I_FFWD : Int;
      I_Outvalue : Int;
   END_VAR
BEGIN

REGION Network 1 (SCL)
   IF "Manage_TC1_2".EnableTC01 AND "Manage_TC1_2".EnableTC02 THEN
       IF NOT "Allarm".TC01_OFR AND NOT "Allarm".TC02_OFR THEN
           "Manage_TC1_2".PID_Ref_Temp := ("Data".Temp_TC01 + "Data".Temp_TC02) / 2;
       ELSIF "Allarm".TC01_OFR THEN
           "Manage_TC1_2".EnableTC01 := FALSE;
       ELSIF "Allarm".TC02_OFR THEN
           "Manage_TC1_2".EnableTC02 := FALSE;
       END_IF;
       "Manage_TC1_2".EmergencyStop := FALSE;
   ELSIF "Manage_TC1_2".EnableTC01 AND NOT "Manage_TC1_2".EnableTC02 THEN
       "Manage_TC1_2".PID_Ref_Temp := "Data".Temp_TC01;
       "Manage_TC1_2".EmergencyStop := FALSE;
       IF "Allarm".TC01_OFR THEN
           "Manage_TC1_2".EnableTC01 := FALSE;
       END_IF;
   ELSIF "Manage_TC1_2".EnableTC02 AND NOT "Manage_TC1_2".EnableTC01 THEN
       "Manage_TC1_2".PID_Ref_Temp := "Data".Temp_TC02;
       "Manage_TC1_2".EmergencyStop := FALSE;
       IF "Allarm".TC01_OFR THEN
           "Manage_TC1_2".EnableTC01 := FALSE;
       END_IF;
   ELSE
       "Manage_TC1_2".EmergencyStop := true;
   END_IF;

   "Allarm".EmergencyStopTC1_2 := "Manage_TC1_2".EmergencyStop;
END_REGION

REGION Network 2 (STL)
   //Converte il setpoint in reale
         L     "Data".TC01_SETPOINT;
         ITD;
         DTR;
         T     #SPValue;

   //Converte il processvalue in reale
         L     "Manage_TC1_2".PID_Ref_Temp;
   //      ITD
   //      DTR
         T     #ProcValue;

   //Converte il manualvalue in reale
         L     "Data".Burner_Panel_SetPoint;
         ITD;
         DTR;
         T     #ManValue;

   //Converte il maxvalue in reale
         L     "Data".Max_PRC_BR1;
         ITD;
         DTR;
         T     #MaxValue;

   //Nega il flag autoburner
         AN    "Flag AutoBurner";
         =     #Manuale;

   //Richiamo FB41 PID_Cont
         CALL  CONT_C, "PID-BURNER"
         ( COM_RST  := FALSE,
           MAN_ON   := #Manuale,
           PVPER_ON := FALSE,
           P_SEL    := TRUE,  //Utilizza parte P
           I_SEL    := TRUE,  //Utilizza parte I
           INT_HOLD := FALSE,
           I_ITL_ON := FALSE,
           D_SEL    := TRUE,  //Utilizza parte D
           CYCLE    := T#1S,  //Intervallo di campionamento
           SP_INT   := #SPValue,  //Valore voluto
           PV_IN    := #ProcValue,  //Valore del processo
           PV_PER   := ,
           MAN      := #ManValue,  //Uscita in manuale
           GAIN     := 1.35,  //coefficiente proporzionale P
           TI       := T#6m,  //Tempo di integrazione I
           TD       := T#5S,  //Tempo del derivatore D
           TM_LAG   := T#5S,  //Tempo di ritardo del componente D
           DEADB_W  := 2.0,  //Banda morta
           LMN_HLM  := #MaxValue,  //Valore superiore uscita
           LMN_LLM  := 5.0,  //Valore inferiore uscita
           PV_FAC   := 1.0,  //Fattore moltiplicativo PROCVALUE
           PV_OFF   := 0.0,  //Fattore offset PROCVALUE
           LMN_FAC  := 1.0,  //Fattore moltiplicativo OUTVALUE
           LMN_OFF  := 0.0,  //Fattore offset OUTVALUE
           I_ITLVAL := ,
           DISV     := ,
           LMN      := #OutValue,
           LMN_PER  := ,
           QLMN_HLM := ,
           QLMN_LLM := ,
           LMN_P    := #TestP,
           LMN_I    := #TestI,
           LMN_D    := #TestD,
           PV       := ,
           ER       :=
         );

   //Converte risultato PID
         L     #OutValue;
         RND;
         T     #I_Outvalue;
END_REGION

REGION Network 3
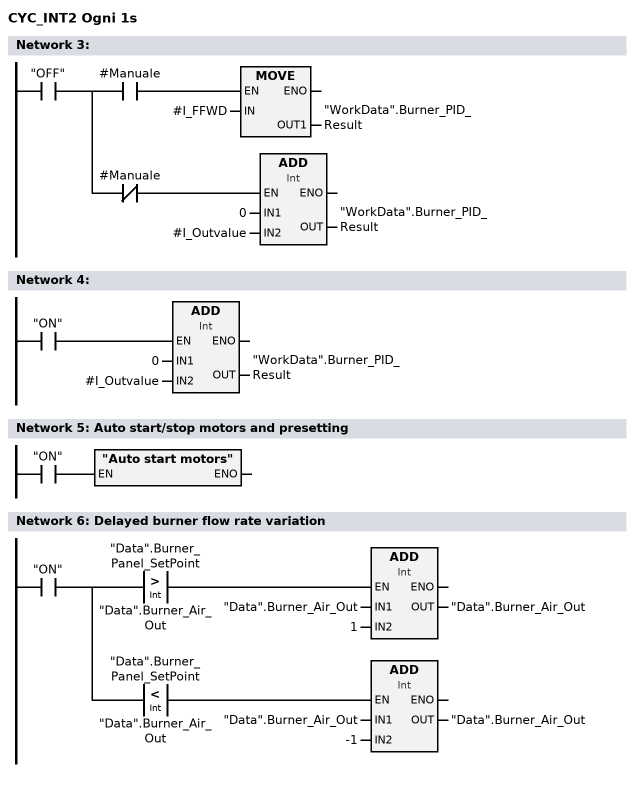
   RUNG wire#powerrail
      Contact( "OFF" )
      wire#w1
      Contact( #Manuale )
      { S7_GenerateENO := "TRUE" } Move(in := #I_FFWD, out1 => "WorkData".Burner_PID_Result)
   END_RUNG
   RUNG wire#w1
      I_Contact( #Manuale )
      { S7_Templates := "SrcType := Int"; S7_GenerateENO := "TRUE" } Add(in1 := 0, in2 := #I_Outvalue, out => "WorkData".Burner_PID_Result)
   END_RUNG
   // the same network as SCL:
   IF "OFF" AND #Manuale THEN "WorkData".Burner_PID_Result := #I_FFWD; END_IF;
   IF "OFF" AND NOT #Manuale THEN "WorkData".Burner_PID_Result := 0 + #I_Outvalue; END_IF;
END_REGION

REGION Network 4
   RUNG wire#powerrail
      Contact( "ON" )
      { S7_Templates := "SrcType := Int"; S7_GenerateENO := "TRUE" } Add(in1 := 0, in2 := #I_Outvalue, out => "WorkData".Burner_PID_Result)
   END_RUNG
   // the same network as SCL:
   IF "ON" THEN "WorkData".Burner_PID_Result := 0 + #I_Outvalue; END_IF;
END_REGION

REGION Network 5: Auto start/stop motors and presetting
   RUNG wire#powerrail
      Contact( "ON" )
      "Auto start motors"()
   END_RUNG
   // the same network as SCL:
   IF "ON" THEN "Auto start motors"(); END_IF;
END_REGION

REGION Network 6: Delayed burner flow rate variation
   RUNG wire#powerrail
      Contact( "ON" )
      wire#w1
      { S7_Templates := "SrcType := Int" } GT_Contact(in1 := "Data".Burner_Panel_SetPoint, in2 := "Data".Burner_Air_Out)
      { S7_Templates := "SrcType := Int"; S7_GenerateENO := "TRUE" } Add(in1 := "Data".Burner_Air_Out, in2 := 1, out => "Data".Burner_Air_Out)
   END_RUNG
   RUNG wire#w1
      { S7_Templates := "SrcType := Int" } LT_Contact(in1 := "Data".Burner_Panel_SetPoint, in2 := "Data".Burner_Air_Out)
      { S7_Templates := "SrcType := Int"; S7_GenerateENO := "TRUE" } Add(in1 := "Data".Burner_Air_Out, in2 := -1, out => "Data".Burner_Air_Out)
   END_RUNG
   // the same network as SCL:
   IF "ON" AND ("Data".Burner_Panel_SetPoint > "Data".Burner_Air_Out) THEN
       "Data".Burner_Air_Out := "Data".Burner_Air_Out + 1;
   END_IF;
   IF "ON" AND ("Data".Burner_Panel_SetPoint < "Data".Burner_Air_Out) THEN
       "Data".Burner_Air_Out := "Data".Burner_Air_Out + (-1);
   END_IF;
END_REGION
END_ORGANIZATION_BLOCK

ORGANIZATION_BLOCK "CYC_INT4 Ogni 200ms"   // OB34, LAD, CyclicInterrupt
TITLE = Ogni 200ms / Every 200ms
{ S7_Optimized_Access := 'FALSE' }
VERSION : 0.1
   VAR_TEMP
      TEMP0 : Byte;
      TEMP1 : Byte;
      TEMP2 : Byte;
      TEMP3 : Byte;
      TEMP4 : Byte;
      TEMP5 : Byte;
      TEMP6 : Int;
      TEMP7 : Int;
      TEMP8 : Int;
      TEMP9 : Date_And_Time;
   END_VAR
BEGIN

REGION Network 1: PER TEST TRENDS / FOR TEST TRENDS
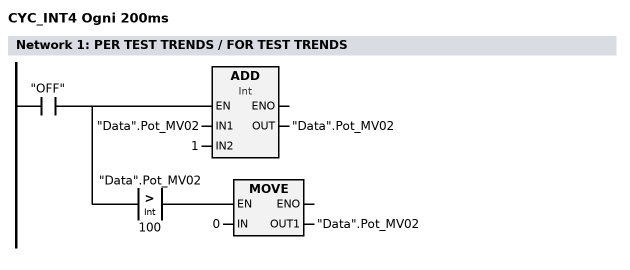
   RUNG wire#powerrail
      Contact( "OFF" )
      wire#w1
      { S7_Templates := "SrcType := Int"; S7_GenerateENO := "TRUE" } Add(in1 := "Data".Pot_MV02, in2 := 1, out => "Data".Pot_MV02)
   END_RUNG
   RUNG wire#w1
      { S7_Templates := "SrcType := Int" } GT_Contact(in1 := "Data".Pot_MV02, in2 := 100)
      { S7_GenerateENO := "TRUE" } Move(in := 0, out1 => "Data".Pot_MV02)
   END_RUNG
   // the same network as SCL:
   IF "OFF" THEN "Data".Pot_MV02 := "Data".Pot_MV02 + 1; END_IF;
   IF "OFF" AND ("Data".Pot_MV02 > 100) THEN "Data".Pot_MV02 := 0; END_IF;
END_REGION
END_ORGANIZATION_BLOCK

ORGANIZATION_BLOCK "CYC_INT5 Ogni 100ms"   // OB35, LAD, CyclicInterrupt
{ S7_Optimized_Access := 'FALSE' }
VERSION : 0.1
   VAR_TEMP
      Real_TC03xMV04 : Real;
      Real_SP_Tc03xMV04 : Real;
      Real_SP_TC03xMV01 : Real;
      Real_O2 : Real;
      Real_SPO2 : Real;
      Real_SPPC01 : Real;
      Real_PC01 : Real;
      VT02Manuale : Bool;
      VT02ManualValue : Real;
      OutVT02 : Real;
      MV05_06_MANUAL : Bool;
      SetMV05_06 : Real;
      OutMV05_06 : Real;
      MV02_MANUAL : Bool;
      SetMV02 : Real;
      OutMV02 : Real;
      MV04_MANUAL : Bool;
      SetMV04 : Real;
      OutMV04 : Real;
      Real_SPPC02 : Real;
      Real_PC02 : Real;
      Real_TC03xMV01 : Real;
   END_VAR
BEGIN

REGION Network 1 (STL)
   //Converte set in reale
         L     "Data".RO01_SETPOINT;  //Prende il valore dal supervisore
         ITD;  //lo converte in DINT
         DTR;  //lo converte in REAL
         T     #Real_SPO2;

   //Converte il valore in reale
         L     "Data".Oxigen_RO01;  //Prende il valore dal supervisore
         ITD;  //lo converte in DINT
         DTR;  //lo converte in REAL
         T     #Real_O2;
END_REGION

REGION Network 2: Controll RO01 moduling MV05 - PID
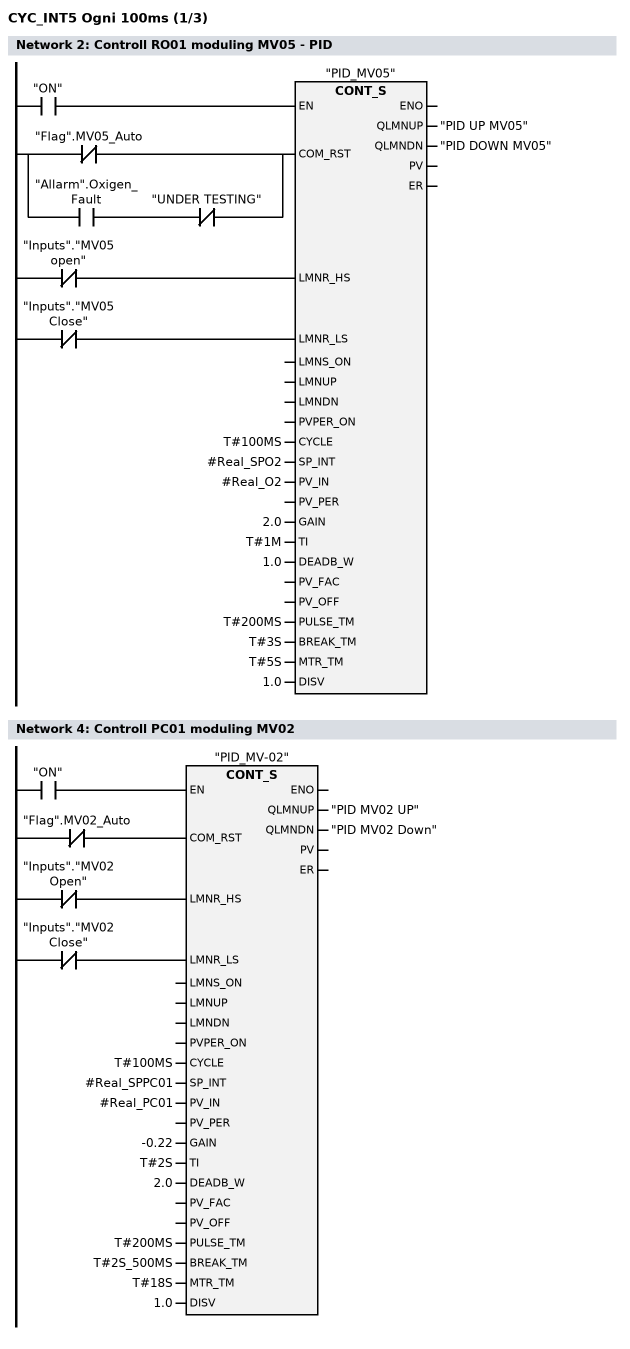
   IF "ON" THEN
       "PID_MV05"(COM_RST := NOT "Flag".MV05_Auto OR ("Allarm".Oxigen_Fault AND NOT "UNDER TESTING"),   // CONT_S
                  LMNR_HS := NOT "Inputs"."MV05 open",
                  LMNR_LS := NOT "Inputs"."MV05 Close",
                  CYCLE := T#100MS,
                  SP_INT := #Real_SPO2,
                  PV_IN := #Real_O2,
                  GAIN := 2.0,
                  TI := T#1M,
                  DEADB_W := 1.0,
                  PULSE_TM := T#200MS,
                  BREAK_TM := T#3S,
                  MTR_TM := T#5S,
                  DISV := 1.0,
                  QLMNUP => "PID UP MV05",
                  QLMNDN => "PID DOWN MV05");
   END_IF;
END_REGION

REGION Network 3 (STL): Controll PC01 moduling MV02 - Converts values into real
   //Converte set in reale
         L     "Data".PSH01_SETPOINT;  //Prende il valore dal supervisore
         ITD;  //lo converte in DINT
         DTR;  //lo converte in REAL
         T     #Real_SPPC01;

   //Converte il valore in reale
         L     "Data".Press_PC01;  //Prende il valore dal supervisore
         ITD;  //lo converte in DINT
         DTR;  //lo converte in REAL
         T     #Real_PC01;
END_REGION

REGION Network 4: Controll PC01 moduling MV02
   IF "ON" THEN
       "PID_MV-02"(COM_RST := NOT "Flag".MV02_Auto,   // CONT_S
                   LMNR_HS := NOT "Inputs"."MV02 Open",
                   LMNR_LS := NOT "Inputs"."MV02 Close",
                   CYCLE := T#100MS,
                   SP_INT := #Real_SPPC01,
                   PV_IN := #Real_PC01,
                   GAIN := -0.22,
                   TI := T#2S,
                   DEADB_W := 2.0,
                   PULSE_TM := T#200MS,
                   BREAK_TM := T#2S_500MS,
                   MTR_TM := T#18S,
                   DISV := 1.0,
                   QLMNUP => "PID MV02 UP",
                   QLMNDN => "PID MV02 Down");
   END_IF;
END_REGION

REGION Network 5
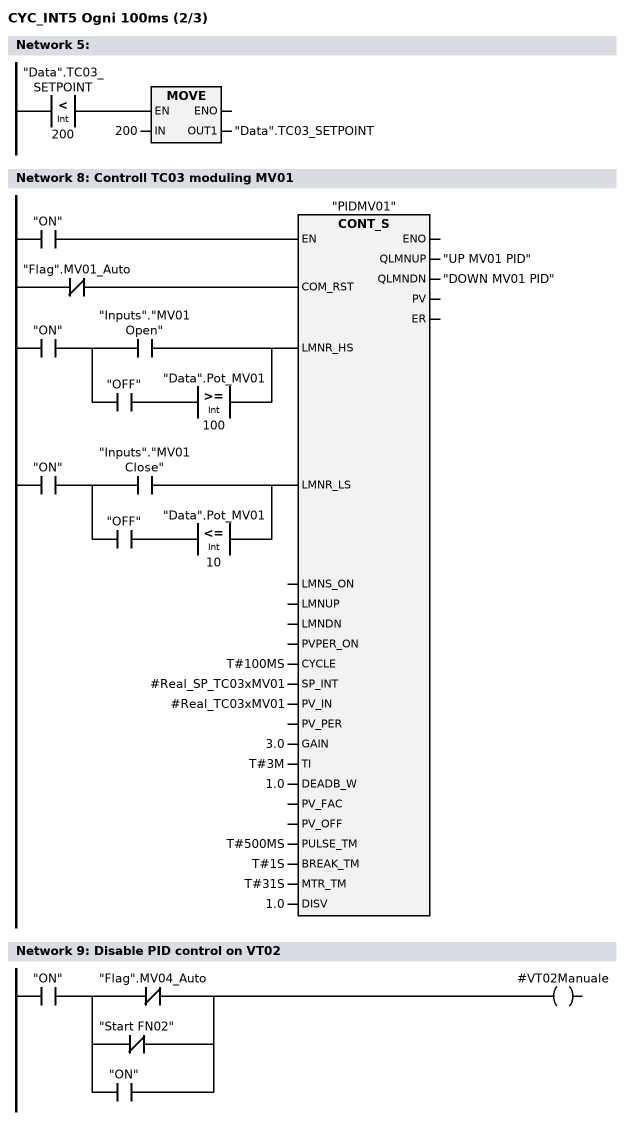
   RUNG wire#powerrail
      { S7_Templates := "SrcType := Int" } LT_Contact(in1 := "Data".TC03_SETPOINT, in2 := 200)
      Move(in := 200, out1 => "Data".TC03_SETPOINT)
   END_RUNG
   // the same network as SCL:
   IF "Data".TC03_SETPOINT < 200 THEN "Data".TC03_SETPOINT := 200; END_IF;
END_REGION

REGION Network 6 (STL): Controll TC03 moduling MV04 - Converts values into real
   //Converte set in reale
         L     "Data".TC03_SETPOINT;  //Prende il valore dal supervisore
         L     -15;  //meno 30°C


         +I;

         ITD;  //lo converte in DINT
         DTR;  //lo converte in REAL
         T     #Real_SP_Tc03xMV04;

   //Converte il valore in reale
         L     "Data".Temp_TC03;  //Prende il valore dal supervisore

         ITD;  //lo converte in DINT
         DTR;  //lo converte in REAL
         T     #Real_TC03xMV04;
END_REGION

REGION Network 7 (STL): Controll TC03 moduling MV01 - Converts values into real
   //Converte set in reale
         L     "Data".TC03_SETPOINT;  //Prende il valore dal supervisore

         L     0;  //meno 0%
         +I;

         ITD;  //lo converte in DINT
         DTR;  //lo converte in REAL
         T     #Real_SP_TC03xMV01;


   //Converte il valore in reale
         L     "Data".Temp_TC03;  //Prende il valore dal supervisore
   //      L     "Data".Temp_T6              //Prende il valore dal supervisore

         ITD;  //lo converte in DINT
         DTR;  //lo converte in REAL
         T     #Real_TC03xMV01;
END_REGION

REGION Network 8: Controll TC03 moduling MV01
   IF "ON" THEN
       "PIDMV01"(COM_RST := NOT "Flag".MV01_Auto,   // CONT_S
                 LMNR_HS := "ON" AND ("Inputs"."MV01 Open" OR ("OFF" AND ("Data".Pot_MV01 >= 100))),
                 LMNR_LS := "ON" AND ("Inputs"."MV01 Close" OR ("OFF" AND ("Data".Pot_MV01 <= 10))),
                 CYCLE := T#100MS,
                 SP_INT := #Real_SP_TC03xMV01,
                 PV_IN := #Real_TC03xMV01,
                 GAIN := 3.0,
                 TI := T#3M,
                 DEADB_W := 1.0,
                 PULSE_TM := T#500MS,
                 BREAK_TM := T#1S,
                 MTR_TM := T#31S,
                 DISV := 1.0,
                 QLMNUP => "UP MV01 PID",
                 QLMNDN => "DOWN MV01 PID");
   END_IF;
END_REGION

REGION Network 9: Disable PID control on VT02
   RUNG wire#powerrail
      Contact( "ON" )
      wire#w1
      I_Contact( "Flag".MV04_Auto )
      wire#w2
      Coil( #VT02Manuale )
   END_RUNG
   RUNG wire#w1
      I_Contact( "Start FN02" )
   END_RUNG wire#w2
   RUNG wire#w1
      Contact( "ON" )
   END_RUNG wire#w2
   // the same network as SCL:
   #VT02Manuale := "ON" AND (NOT "Flag".MV04_Auto OR NOT "Start FN02" OR "ON");
END_REGION

REGION Network 10 (STL): The temperature of TC03 Moduling the speed of VT02
   //Converte il manualvalue in reale normalizzandolo in 100..0
         L     0;
         L     "Data".Set_Perc_VT02;
         +I;
         ITD;
         DTR;
         T     #VT02ManualValue;

   //Richiamo FB41 PID_Cont
         CALL  CONT_C, "PID_VT02"
         ( COM_RST  := FALSE,
           MAN_ON   := #VT02Manuale,
           PVPER_ON := FALSE,
           P_SEL    := TRUE,  //Utilizza parte P
           I_SEL    := TRUE,  //Utilizza parte I
           INT_HOLD := ,
           I_ITL_ON := ,
           D_SEL    := FALSE,  //Utilizza parte D
           CYCLE    := T#100MS,  //Intervallo di campionamento
           SP_INT   := #Real_SP_Tc03xMV04,  //Valore voluto
           PV_IN    := #Real_TC03xMV04,  //Valore del processo
           PV_PER   := ,
           MAN      := #VT02ManualValue,  //Uscita in manuale
           GAIN     := "DATA_PID".GAIN_FN02,  //coefficiente proporzionale P
           TI       := "DATA_PID".TI_FN02,  //Tempo di integrazione I
           TD       := T#1M,  //Tempo del derivatore D
           TM_LAG   := T#1M,  //Tempo di ritardo del componente D
           DEADB_W  := 1.5,  //Banda morta
           LMN_HLM  := 100.0,  //Valore superiore uscita (50%)
           LMN_LLM  := 35.0,  //Valore inferiore uscita (100%)
           PV_FAC   := ,
           PV_OFF   := ,
           LMN_FAC  := 1.0,  //Fattore moltiplicativo OUTVALUE
           LMN_OFF  := 0.0,  //Fattore offset OUTVALUE
           I_ITLVAL := ,
           DISV     := 1.0,  //Fattore di disturbo
           LMN      := #OutVT02,  //Uscita regolante
           LMN_PER  := ,
           QLMN_HLM := ,
           QLMN_LLM := ,
           LMN_P    := ,
           LMN_I    := ,
           LMN_D    := ,
           PV       := ,
           ER       :=
         );

   //Converte risultato PID 0..100 -> 100..0
         L     0.0;
         L     #OutVT02;
         +R;
         RND;
         T     "Data".Set_Perc_VT02;
END_REGION

REGION Network 11 (STL): Control PC02 Moduling MV03 - Convert values in real
   //Converte set in reale
         L     "Data".PSH02_SETPOINT;  //Prende il valore dal supervisore
         ITD;  //lo converte in DINT
         DTR;  //lo converte in REAL
         T     #Real_SPPC02;

   //Converte il valore in reale
         L     "Data".PSH_02;  //Prende il valore dal supervisore
         ITD;  //lo converte in DINT
         DTR;  //lo converte in REAL
         T     #Real_PC02;
END_REGION

REGION Network 12: Control PC02 Moduling MV03 - NOT USED
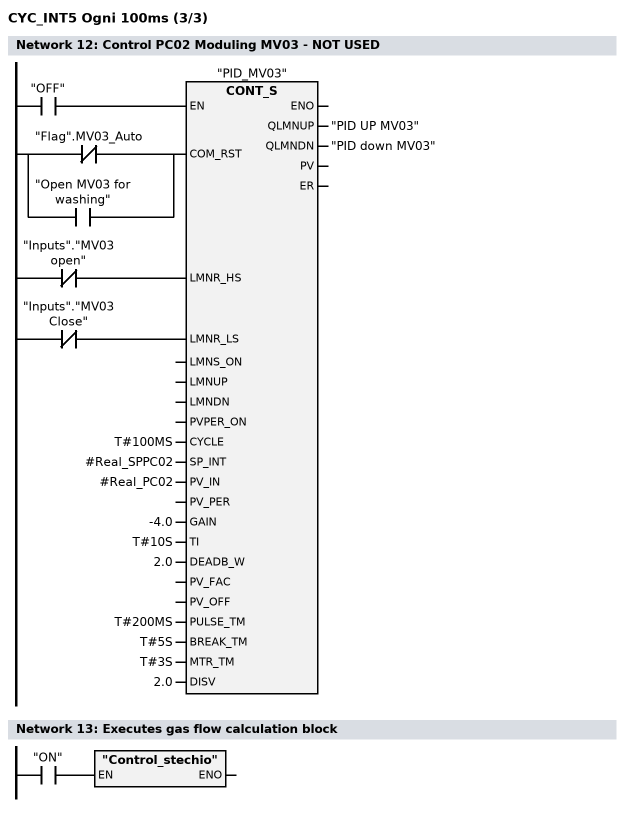
   IF "OFF" THEN
       "PID_MV03"(COM_RST := NOT "Flag".MV03_Auto OR "Open MV03 for washing",   // CONT_S
                  LMNR_HS := NOT "Inputs"."MV03 open",
                  LMNR_LS := NOT "Inputs"."MV03 Close",
                  CYCLE := T#100MS,
                  SP_INT := #Real_SPPC02,
                  PV_IN := #Real_PC02,
                  GAIN := -4.0,
                  TI := T#10S,
                  DEADB_W := 2.0,
                  PULSE_TM := T#200MS,
                  BREAK_TM := T#5S,
                  MTR_TM := T#3S,
                  DISV := 2.0,
                  QLMNUP => "PID UP MV03",
                  QLMNDN => "PID down MV03");
   END_IF;
END_REGION

REGION Network 13: Executes gas flow calculation block
   RUNG wire#powerrail
      Contact( "ON" )
      "Control_stechio"()
   END_RUNG
   // the same network as SCL:
   IF "ON" THEN "Control_stechio"(); END_IF;
END_REGION
END_ORGANIZATION_BLOCK

ORGANIZATION_BLOCK "I/O_FLT1"   // OB82, LAD, DiagnosticErrorInterrupt
TITLE = "I/O Point Fault"
{ S7_Optimized_Access := 'FALSE' }
VERSION : 0.1
   VAR_TEMP
      OB82_EV_CLASS : Byte;   // 16#39, Event class 3, Entering event state, Internal fault event
      OB82_FLT_ID : Byte;   // 16#XX, Fault identifcation code
      OB82_PRIORITY : Byte;   // Priority of OB Execution
      OB82_OB_NUMBR : Byte;   // 82 (Organization block 82, OB82)
      OB82_RESERVED_1 : Byte;   // Reserved for system
      OB82_IO_FLAG : Byte;   // Input (01010100), Output (01010101)
      OB82_MDL_ADDR : Word;   // Base address of module with fault
      OB82_MDL_DEFECT : Bool;   // Module defective
      OB82_INT_FAULT : Bool;   // Internal fault
      OB82_EXT_FAULT : Bool;   // External fault
      OB82_PNT_INFO : Bool;   // Point information
      OB82_EXT_VOLTAGE : Bool;   // External voltage low
      OB82_FLD_CONNCTR : Bool;   // Field wiring connector missing
      OB82_NO_CONFIG : Bool;   // Module has no configuration data
      OB82_CONFIG_ERR : Bool;   // Module has configuration error
      OB82_MDL_TYPE : Byte;   // Type of module
      OB82_SUB_MDL_ERR : Bool;   // Sub-Module is missing or has error
      OB82_COMM_FAULT : Bool;   // Communication fault
      OB82_MDL_STOP : Bool;   // Module is stopped
      OB82_WTCH_DOG_FLT : Bool;   // Watch dog timer stopped module
      OB82_INT_PS_FLT : Bool;   // Internal power supply fault
      OB82_PRIM_BATT_FLT : Bool;   // Primary battery is in fault
      OB82_BCKUP_BATT_FLT : Bool;   // Backup battery is in fault
      OB82_RESERVED_2 : Bool;   // Reserved for system
      OB82_RACK_FLT : Bool;   // Rack fault, only for bus interface module
      OB82_PROC_FLT : Bool;   // Processor fault
      OB82_EPROM_FLT : Bool;   // EPROM fault
      OB82_RAM_FLT : Bool;   // RAM fault
      OB82_ADU_FLT : Bool;   // ADU fault
      OB82_FUSE_FLT : Bool;   // Fuse fault
      OB82_HW_INTR_FLT : Bool;   // Hardware interupt input in fault
      OB82_RESERVED_3 : Bool;   // Reserved for system
      OB82_DATE_TIME : Date_And_Time;   // Date and time OB82 started
   END_VAR
BEGIN

REGION Network 1
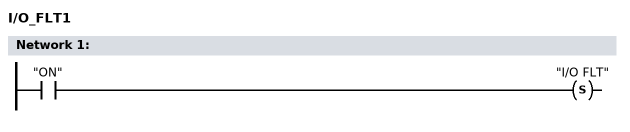
   RUNG wire#powerrail
      Contact( "ON" )
      S_Coil( "I/O FLT" )
   END_RUNG
   // the same network as SCL:
   IF "ON" THEN "I/O FLT" := TRUE; END_IF;
END_REGION
END_ORGANIZATION_BLOCK

ORGANIZATION_BLOCK "RACK_FLT"   // OB86, LAD, RackStationFailure
TITLE = "Loss Of Rack Fault"
{ S7_Optimized_Access := 'FALSE' }
VERSION : 0.1
// Questo OB viene lanciato se un rack è: disconnesso, oppure un modulo di un rack 
// è disconnesso
// This OB is launched if a rack is: disconnected, or a module of a rack
   VAR_TEMP
      OB86_EV_CLASS : Byte;   // 16#38/39 Event class 3
      OB86_FLT_ID : Byte;   // 16#C1/C4/C5, Fault identifcation code
      OB86_PRIORITY : Byte;   // Priority of OB Execution
      OB86_OB_NUMBR : Byte;   // 86 (Organization block 86, OB86)
      OB86_RESERVED_1 : Byte;   // Reserved for system
      OB86_RESERVED_2 : Byte;   // Reserved for system
      OB86_MDL_ADDR : Word;   // Base address of IM module in rack with fault
      OB86_RACKS_FLTD : Array[0..31] of Bool;
      OB86_DATE_TIME : Date_And_Time;   // Date and time OB86 started
   END_VAR
BEGIN

REGION Network 1
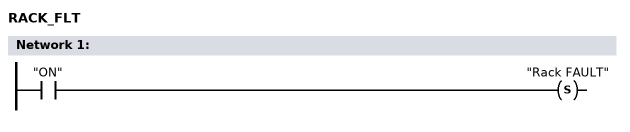
   RUNG wire#powerrail
      Contact( "ON" )
      S_Coil( "Rack FAULT" )
   END_RUNG
   // the same network as SCL:
   IF "ON" THEN "Rack FAULT" := TRUE; END_IF;
END_REGION
END_ORGANIZATION_BLOCK

ORGANIZATION_BLOCK "Startup only"   // OB100, LAD, Startup
TITLE = Power up - Start up
{ S7_Optimized_Access := 'FALSE' }
VERSION : 0.1
   VAR_TEMP
      TEMP0 : Byte;
      TEMP1 : Byte;
      TEMP2 : Byte;
      TEMP3 : Byte;
      TEMP4 : Byte;
      TEMP5 : Byte;
      TEMP6 : Word;
      TEMP7 : DWord;
      TEMP8 : Date_And_Time;
      App01 : Int;
   END_VAR
BEGIN

REGION Network 1 (STL): Special flag initialization
         SET;
         S     "ON";
         CLR;
         S     "OFF";
END_REGION

REGION Network 2: reset all flag start motors
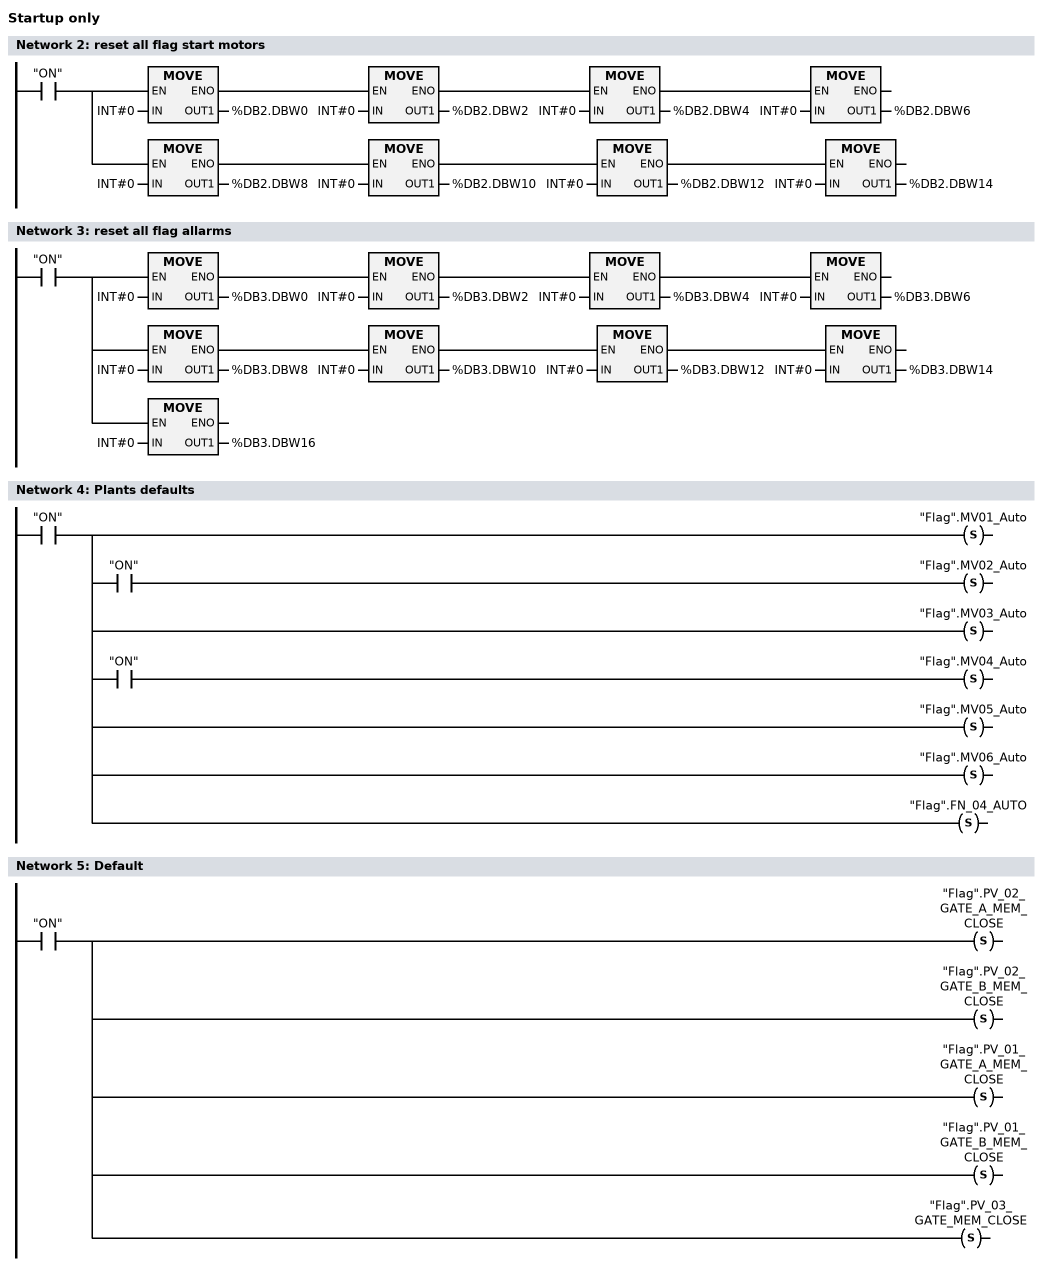
   RUNG wire#powerrail
      Contact( "ON" )
      wire#w1
      { S7_GenerateENO := "TRUE" } Move(in := INT#0, out1 => %DB2.DBW0)
      { S7_GenerateENO := "TRUE" } Move(in := INT#0, out1 => %DB2.DBW2)
      { S7_GenerateENO := "TRUE" } Move(in := INT#0, out1 => %DB2.DBW4)
      { S7_GenerateENO := "TRUE" } Move(in := INT#0, out1 => %DB2.DBW6)
   END_RUNG
   RUNG wire#w1
      { S7_GenerateENO := "TRUE" } Move(in := INT#0, out1 => %DB2.DBW8)
      { S7_GenerateENO := "TRUE" } Move(in := INT#0, out1 => %DB2.DBW10)
      { S7_GenerateENO := "TRUE" } Move(in := INT#0, out1 => %DB2.DBW12)
      { S7_GenerateENO := "TRUE" } Move(in := INT#0, out1 => %DB2.DBW14)
   END_RUNG
   // the same network as SCL:
   // ENO of a box is taken as its EN; it also drops when the box reports an error
   IF "ON" THEN
       %DB2.DBW0 := INT#0;
       %DB2.DBW2 := INT#0;
       %DB2.DBW4 := INT#0;
       %DB2.DBW6 := INT#0;
       %DB2.DBW8 := INT#0;
       %DB2.DBW10 := INT#0;
       %DB2.DBW12 := INT#0;
       %DB2.DBW14 := INT#0;
   END_IF;
END_REGION

REGION Network 3: reset all flag allarms
   RUNG wire#powerrail
      Contact( "ON" )
      wire#w1
      { S7_GenerateENO := "TRUE" } Move(in := INT#0, out1 => %DB3.DBW0)
      { S7_GenerateENO := "TRUE" } Move(in := INT#0, out1 => %DB3.DBW2)
      { S7_GenerateENO := "TRUE" } Move(in := INT#0, out1 => %DB3.DBW4)
      { S7_GenerateENO := "TRUE" } Move(in := INT#0, out1 => %DB3.DBW6)
   END_RUNG
   RUNG wire#w1
      { S7_GenerateENO := "TRUE" } Move(in := INT#0, out1 => %DB3.DBW8)
      { S7_GenerateENO := "TRUE" } Move(in := INT#0, out1 => %DB3.DBW10)
      { S7_GenerateENO := "TRUE" } Move(in := INT#0, out1 => %DB3.DBW12)
      { S7_GenerateENO := "TRUE" } Move(in := INT#0, out1 => %DB3.DBW14)
   END_RUNG
   RUNG wire#w1
      { S7_GenerateENO := "TRUE" } Move(in := INT#0, out1 => %DB3.DBW16)
   END_RUNG
   // the same network as SCL:
   // ENO of a box is taken as its EN; it also drops when the box reports an error
   IF "ON" THEN
       %DB3.DBW0 := INT#0;
       %DB3.DBW2 := INT#0;
       %DB3.DBW4 := INT#0;
       %DB3.DBW6 := INT#0;
       %DB3.DBW8 := INT#0;
       %DB3.DBW10 := INT#0;
       %DB3.DBW12 := INT#0;
       %DB3.DBW14 := INT#0;
       %DB3.DBW16 := INT#0;
   END_IF;
END_REGION

REGION Network 4: Plants defaults
   RUNG wire#powerrail
      Contact( "ON" )
      wire#w1
      S_Coil( "Flag".MV01_Auto )
   END_RUNG
   RUNG wire#w1
      Contact( "ON" )
      S_Coil( "Flag".MV02_Auto )
   END_RUNG
   RUNG wire#w1
      S_Coil( "Flag".MV03_Auto )
   END_RUNG
   RUNG wire#w1
      Contact( "ON" )
      S_Coil( "Flag".MV04_Auto )
   END_RUNG
   RUNG wire#w1
      S_Coil( "Flag".MV05_Auto )
   END_RUNG
   RUNG wire#w1
      S_Coil( "Flag".MV06_Auto )
   END_RUNG
   RUNG wire#w1
      S_Coil( "Flag".FN_04_AUTO )
   END_RUNG
   // the same network as SCL:
   IF "ON" THEN "Flag".MV01_Auto := TRUE; END_IF;
   IF "ON" AND "ON" THEN "Flag".MV02_Auto := TRUE; END_IF;
   IF "ON" THEN "Flag".MV03_Auto := TRUE; END_IF;
   IF "ON" AND "ON" THEN "Flag".MV04_Auto := TRUE; END_IF;
   IF "ON" THEN
       "Flag".MV05_Auto := TRUE;
       "Flag".MV06_Auto := TRUE;
       "Flag".FN_04_AUTO := TRUE;
   END_IF;
END_REGION

REGION Network 5: Default
   RUNG wire#powerrail
      Contact( "ON" )
      wire#w1
      S_Coil( "Flag".PV_02_GATE_A_MEM_CLOSE )
   END_RUNG
   RUNG wire#w1
      S_Coil( "Flag".PV_02_GATE_B_MEM_CLOSE )
   END_RUNG
   RUNG wire#w1
      S_Coil( "Flag".PV_01_GATE_A_MEM_CLOSE )
   END_RUNG
   RUNG wire#w1
      S_Coil( "Flag".PV_01_GATE_B_MEM_CLOSE )
   END_RUNG
   RUNG wire#w1
      S_Coil( "Flag".PV_03_GATE_MEM_CLOSE )
   END_RUNG
   // the same network as SCL:
   IF "ON" THEN
       "Flag".PV_02_GATE_A_MEM_CLOSE := TRUE;
       "Flag".PV_02_GATE_B_MEM_CLOSE := TRUE;
       "Flag".PV_01_GATE_A_MEM_CLOSE := TRUE;
       "Flag".PV_01_GATE_B_MEM_CLOSE := TRUE;
       "Flag".PV_03_GATE_MEM_CLOSE := TRUE;
   END_IF;
END_REGION
END_ORGANIZATION_BLOCK

ORGANIZATION_BLOCK "PROG_ERR"   // OB121, LAD, ProgrammingError
TITLE = "Programming Error"
{ S7_Optimized_Access := 'FALSE' }
VERSION : 0.1
   VAR_TEMP
      OB121_EV_CLASS : Byte;   // 16#25, Event class 2, Entering event state, Internal fault event
      OB121_SW_FLT : Byte;   // 16#XX Software programming fault
      OB121_PRIORITY : Byte;   // Priority of OB Execution
      OB121_OB_NUMBR : Byte;   // 121 (Organization block 121, OB121)
      OB121_BLK_TYPE : Byte;   // 16#88/8A/8B/8C/8E Type of block fault occured in
      OB121_RESERVED_1 : Byte;   // Reserved for system
      OB121_FLT_REG : Word;   // 16#XX Specific register that caused fault
      OB121_BLK_NUM : Word;   // Number of block that programming fault occured in
      OB121_PRG_ADDR : Word;   // Address in block where programming fault occured
      OB121_DATE_TIME : Date_And_Time;   // Date and time OB121 started
   END_VAR
BEGIN

REGION Network 1
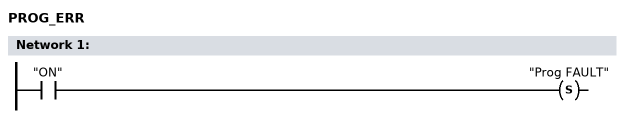
   RUNG wire#powerrail
      Contact( "ON" )
      S_Coil( "Prog FAULT" )
   END_RUNG
   // the same network as SCL:
   IF "ON" THEN "Prog FAULT" := TRUE; END_IF;
END_REGION
END_ORGANIZATION_BLOCK

ORGANIZATION_BLOCK "MOD_ERR"   // OB122, LAD, IOAccessError
TITLE = "Module Access Error"
{ S7_Optimized_Access := 'FALSE' }
VERSION : 0.1
   VAR_TEMP
      OB122_EV_CLASS : Byte;   // 16#29, Event class 2, Entering event state, Internal fault event
      OB122_SW_FLT : Byte;   // 16#XX Software error code
      OB122_PRIORITY : Byte;   // Priority of OB Execution
      OB122_OB_NUMBR : Byte;   // 122 (Organization block 122, OB122)
      OB122_BLK_TYPE : Byte;   // 16#88/8C/8E Type of block fault occured in
      OB122_MEM_AREA : Byte;   // Memory area where access error occured
      OB122_MEM_ADDR : Word;   // Memory address where access error occured
      OB122_BLK_NUM : Word;   // Block number in which error occured
      OB122_PRG_ADDR : Word;   // Program address where error occured
      OB122_DATE_TIME : Date_And_Time;   // Date and time OB1 started
   END_VAR
BEGIN

REGION Network 1
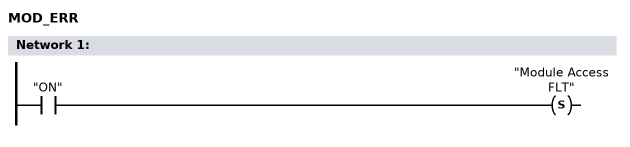
   RUNG wire#powerrail
      Contact( "ON" )
      S_Coil( "Module Access FLT" )
   END_RUNG
   // the same network as SCL:
   IF "ON" THEN "Module Access FLT" := TRUE; END_IF;
END_REGION
END_ORGANIZATION_BLOCK

// folder: FOR HMI

FUNCTION "HMI Standard Motors" : Void   // FC1, LAD
{ S7_Optimized_Access := 'TRUE' }
VERSION : 0.1
   VAR_INPUT
      Ingresso_run : Bool;
      Allarme1 : Bool;
      Allarme2 : Bool;
      Allarme3 : Bool;
      Allarme4 : Bool;
      Allarme5 : Bool;
   END_VAR
   VAR_OUTPUT
      Risposta : Bool;
      Comulativo_allarmi : Bool;
   END_VAR
BEGIN

REGION Network 1
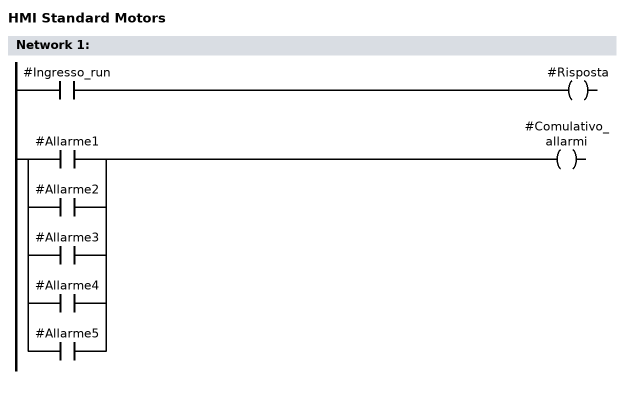
   RUNG wire#powerrail
      Contact( #Ingresso_run )
      Coil( #Risposta )
   END_RUNG
   RUNG wire#powerrail
      Contact( #Allarme1 )
      wire#w1
      Coil( #Comulativo_allarmi )
   END_RUNG
   RUNG wire#powerrail
      Contact( #Allarme2 )
   END_RUNG wire#w1
   RUNG wire#powerrail
      Contact( #Allarme3 )
   END_RUNG wire#w1
   RUNG wire#powerrail
      Contact( #Allarme4 )
   END_RUNG wire#w1
   RUNG wire#powerrail
      Contact( #Allarme5 )
   END_RUNG wire#w1
   // the same network as SCL:
   #Risposta := #Ingresso_run;
   #Comulativo_allarmi := #Allarme1 OR #Allarme2 OR #Allarme3 OR #Allarme4 OR #Allarme5;
END_REGION
END_FUNCTION

FUNCTION "HMI Standard Motorized Valve" : Void   // FC10, LAD
{ S7_Optimized_Access := 'TRUE' }
VERSION : 0.1
   VAR_INPUT
      Ingresso_run_Opening : Bool;
      Ingresso_run_Closing : Bool;
      Allarme1 : Bool;
      Allarme2 : Bool;
      Allarme3 : Bool;
      Allarme4 : Bool;
      Allarme5 : Bool;
      Limit_switch_Open : Bool;
      Limiti_Switch_Close : Bool;
   END_VAR
   VAR_OUTPUT
      Risposta_Opening : Bool;
      Risposta_Closing : Bool;
      Limit_Switch_Open_HMI : Bool;
      Limit_Switch_Close_HMI : Bool;
      Comulativo_allarmi : Bool;
   END_VAR
BEGIN

REGION Network 1
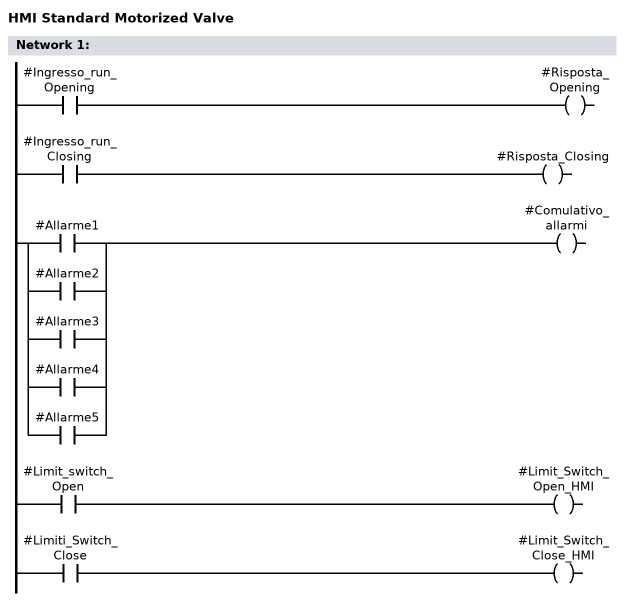
   RUNG wire#powerrail
      Contact( #Ingresso_run_Opening )
      Coil( #Risposta_Opening )
   END_RUNG
   RUNG wire#powerrail
      Contact( #Ingresso_run_Closing )
      Coil( #Risposta_Closing )
   END_RUNG
   RUNG wire#powerrail
      Contact( #Allarme1 )
      wire#w1
      Coil( #Comulativo_allarmi )
   END_RUNG
   RUNG wire#powerrail
      Contact( #Allarme2 )
   END_RUNG wire#w1
   RUNG wire#powerrail
      Contact( #Allarme3 )
   END_RUNG wire#w1
   RUNG wire#powerrail
      Contact( #Allarme4 )
   END_RUNG wire#w1
   RUNG wire#powerrail
      Contact( #Allarme5 )
   END_RUNG wire#w1
   RUNG wire#powerrail
      Contact( #Limit_switch_Open )
      Coil( #Limit_Switch_Open_HMI )
   END_RUNG
   RUNG wire#powerrail
      Contact( #Limiti_Switch_Close )
      Coil( #Limit_Switch_Close_HMI )
   END_RUNG
   // the same network as SCL:
   #Risposta_Opening := #Ingresso_run_Opening;
   #Risposta_Closing := #Ingresso_run_Closing;
   #Comulativo_allarmi := #Allarme1 OR #Allarme2 OR #Allarme3 OR #Allarme4 OR #Allarme5;
   #Limit_Switch_Open_HMI := #Limit_switch_Open;
   #Limit_Switch_Close_HMI := #Limiti_Switch_Close;
END_REGION
END_FUNCTION

FUNCTION "HMI" : Void   // FC11, LAD
{ S7_Optimized_Access := 'TRUE' }
VERSION : 0.1
BEGIN

REGION Network 1: BC01
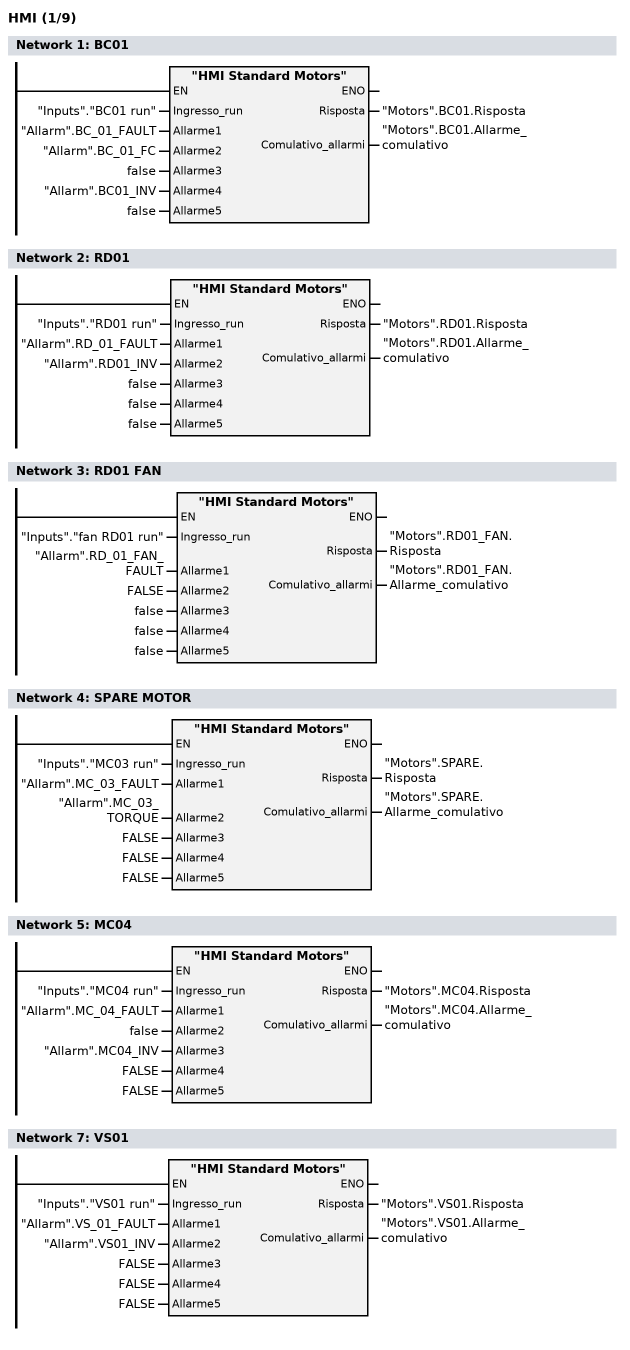
   RUNG wire#powerrail
      "HMI Standard Motors"(Ingresso_run := "Inputs"."BC01 run", Allarme1 := "Allarm".BC_01_FAULT, Allarme2 := "Allarm".BC_01_FC, Allarme3 := false, Allarme4 := "Allarm".BC01_INV, Allarme5 := false, Risposta => "Motors".BC01.Risposta, Comulativo_allarmi => "Motors".BC01.Allarme_comulativo)
   END_RUNG
   // the same network as SCL:
   "HMI Standard Motors"(Ingresso_run := "Inputs"."BC01 run",
                         Allarme1 := "Allarm".BC_01_FAULT,
                         Allarme2 := "Allarm".BC_01_FC,
                         Allarme3 := false,
                         Allarme4 := "Allarm".BC01_INV,
                         Allarme5 := false,
                         Risposta => "Motors".BC01.Risposta,
                         Comulativo_allarmi => "Motors".BC01.Allarme_comulativo);
END_REGION

REGION Network 2: RD01
   RUNG wire#powerrail
      "HMI Standard Motors"(Ingresso_run := "Inputs"."RD01 run", Allarme1 := "Allarm".RD_01_FAULT, Allarme2 := "Allarm".RD01_INV, Allarme3 := false, Allarme4 := false, Allarme5 := false, Risposta => "Motors".RD01.Risposta, Comulativo_allarmi => "Motors".RD01.Allarme_comulativo)
   END_RUNG
   // the same network as SCL:
   "HMI Standard Motors"(Ingresso_run := "Inputs"."RD01 run",
                         Allarme1 := "Allarm".RD_01_FAULT,
                         Allarme2 := "Allarm".RD01_INV,
                         Allarme3 := false,
                         Allarme4 := false,
                         Allarme5 := false,
                         Risposta => "Motors".RD01.Risposta,
                         Comulativo_allarmi => "Motors".RD01.Allarme_comulativo);
END_REGION

REGION Network 3: RD01 FAN
   RUNG wire#powerrail
      "HMI Standard Motors"(Ingresso_run := "Inputs"."fan RD01 run", Allarme1 := "Allarm".RD_01_FAN_FAULT, Allarme2 := FALSE, Allarme3 := false, Allarme4 := false, Allarme5 := false, Risposta => "Motors".RD01_FAN.Risposta, Comulativo_allarmi => "Motors".RD01_FAN.Allarme_comulativo)
   END_RUNG
   // the same network as SCL:
   "HMI Standard Motors"(Ingresso_run := "Inputs"."fan RD01 run",
                         Allarme1 := "Allarm".RD_01_FAN_FAULT,
                         Allarme2 := FALSE,
                         Allarme3 := false,
                         Allarme4 := false,
                         Allarme5 := false,
                         Risposta => "Motors".RD01_FAN.Risposta,
                         Comulativo_allarmi => "Motors".RD01_FAN.Allarme_comulativo);
END_REGION

REGION Network 4: SPARE MOTOR
   RUNG wire#powerrail
      "HMI Standard Motors"(Ingresso_run := "Inputs"."MC03 run", Allarme1 := "Allarm".MC_03_FAULT, Allarme2 := "Allarm".MC_03_TORQUE, Allarme3 := FALSE, Allarme4 := FALSE, Allarme5 := FALSE, Risposta => "Motors".SPARE.Risposta, Comulativo_allarmi => "Motors".SPARE.Allarme_comulativo)
   END_RUNG
   // the same network as SCL:
   "HMI Standard Motors"(Ingresso_run := "Inputs"."MC03 run",
                         Allarme1 := "Allarm".MC_03_FAULT,
                         Allarme2 := "Allarm".MC_03_TORQUE,
                         Allarme3 := FALSE,
                         Allarme4 := FALSE,
                         Allarme5 := FALSE,
                         Risposta => "Motors".SPARE.Risposta,
                         Comulativo_allarmi => "Motors".SPARE.Allarme_comulativo);
END_REGION

REGION Network 5: MC04
   RUNG wire#powerrail
      "HMI Standard Motors"(Ingresso_run := "Inputs"."MC04 run", Allarme1 := "Allarm".MC_04_FAULT, Allarme2 := false, Allarme3 := "Allarm".MC04_INV, Allarme4 := FALSE, Allarme5 := FALSE, Risposta => "Motors".MC04.Risposta, Comulativo_allarmi => "Motors".MC04.Allarme_comulativo)
   END_RUNG
   // the same network as SCL:
   "HMI Standard Motors"(Ingresso_run := "Inputs"."MC04 run",
                         Allarme1 := "Allarm".MC_04_FAULT,
                         Allarme2 := false,
                         Allarme3 := "Allarm".MC04_INV,
                         Allarme4 := FALSE,
                         Allarme5 := FALSE,
                         Risposta => "Motors".MC04.Risposta,
                         Comulativo_allarmi => "Motors".MC04.Allarme_comulativo);
END_REGION

REGION Network 6: MC05 DELETED
END_REGION

REGION Network 7: VS01
   RUNG wire#powerrail
      "HMI Standard Motors"(Ingresso_run := "Inputs"."VS01 run", Allarme1 := "Allarm".VS_01_FAULT, Allarme2 := "Allarm".VS01_INV, Allarme3 := FALSE, Allarme4 := FALSE, Allarme5 := FALSE, Risposta => "Motors".VS01.Risposta, Comulativo_allarmi => "Motors".VS01.Allarme_comulativo)
   END_RUNG
   // the same network as SCL:
   "HMI Standard Motors"(Ingresso_run := "Inputs"."VS01 run",
                         Allarme1 := "Allarm".VS_01_FAULT,
                         Allarme2 := "Allarm".VS01_INV,
                         Allarme3 := FALSE,
                         Allarme4 := FALSE,
                         Allarme5 := FALSE,
                         Risposta => "Motors".VS01.Risposta,
                         Comulativo_allarmi => "Motors".VS01.Allarme_comulativo);
END_REGION

REGION Network 8: SC12 DELETED
END_REGION

REGION Network 9: AUXILIARY INVERTER
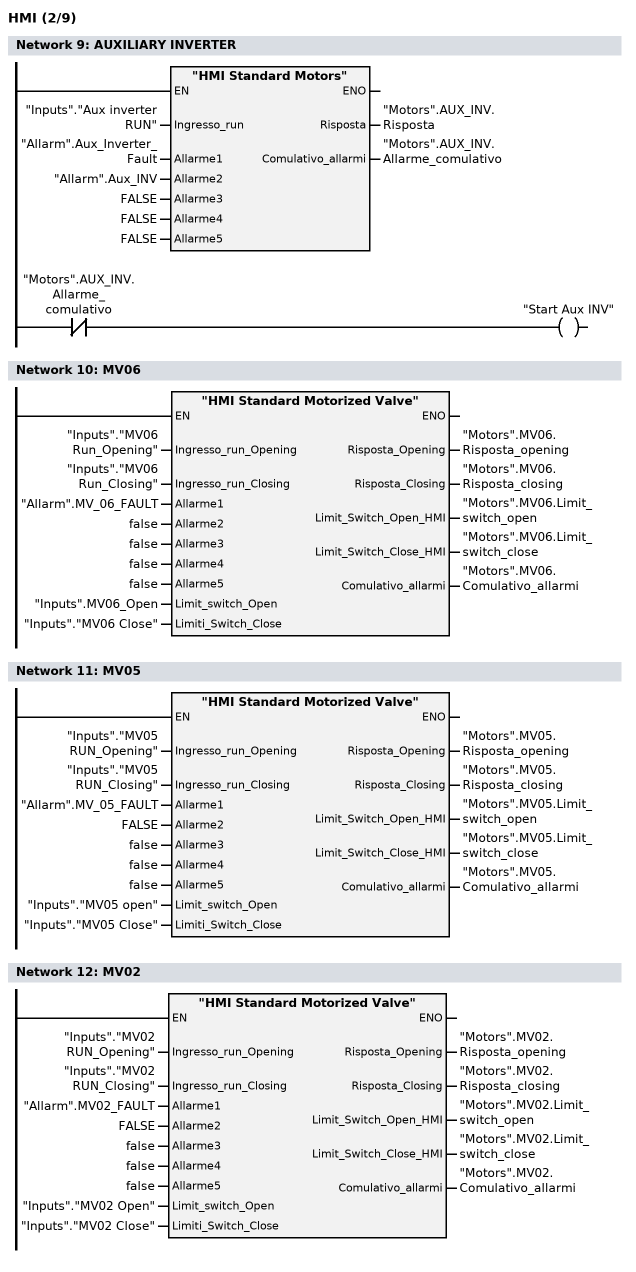
   RUNG wire#powerrail
      "HMI Standard Motors"(Ingresso_run := "Inputs"."Aux inverter RUN", Allarme1 := "Allarm".Aux_Inverter_Fault, Allarme2 := "Allarm".Aux_INV, Allarme3 := FALSE, Allarme4 := FALSE, Allarme5 := FALSE, Risposta => "Motors".AUX_INV.Risposta, Comulativo_allarmi => "Motors".AUX_INV.Allarme_comulativo)
   END_RUNG
   RUNG wire#powerrail
      I_Contact( "Motors".AUX_INV.Allarme_comulativo )
      Coil( "Start Aux INV" )
   END_RUNG
   // the same network as SCL:
   "HMI Standard Motors"(Ingresso_run := "Inputs"."Aux inverter RUN",
                         Allarme1 := "Allarm".Aux_Inverter_Fault,
                         Allarme2 := "Allarm".Aux_INV,
                         Allarme3 := FALSE,
                         Allarme4 := FALSE,
                         Allarme5 := FALSE,
                         Risposta => "Motors".AUX_INV.Risposta,
                         Comulativo_allarmi => "Motors".AUX_INV.Allarme_comulativo);
   "Start Aux INV" := NOT "Motors".AUX_INV.Allarme_comulativo;
END_REGION

REGION Network 10: MV06
   RUNG wire#powerrail
      "HMI Standard Motorized Valve"(Ingresso_run_Opening := "Inputs"."MV06 Run_Opening", Ingresso_run_Closing := "Inputs"."MV06 Run_Closing", Allarme1 := "Allarm".MV_06_FAULT, Allarme2 := false, Allarme3 := false, Allarme4 := false, Allarme5 := false, Limit_switch_Open := "Inputs".MV06_Open, Limiti_Switch_Close := "Inputs"."MV06 Close", Risposta_Opening => "Motors".MV06.Risposta_opening, Risposta_Closing => "Motors".MV06.Risposta_closing, Limit_Switch_Open_HMI => "Motors".MV06.Limit_switch_open, Limit_Switch_Close_HMI => "Motors".MV06.Limit_switch_close, Comulativo_allarmi => "Motors".MV06.Comulativo_allarmi)
   END_RUNG
   // the same network as SCL:
   "HMI Standard Motorized Valve"(Ingresso_run_Opening := "Inputs"."MV06 Run_Opening",
                           Ingresso_run_Closing := "Inputs"."MV06 Run_Closing",
                           Allarme1 := "Allarm".MV_06_FAULT,
                           Allarme2 := false,
                           Allarme3 := false,
                           Allarme4 := false,
                           Allarme5 := false,
                           Limit_switch_Open := "Inputs".MV06_Open,
                           Limiti_Switch_Close := "Inputs"."MV06 Close",
                           Risposta_Opening => "Motors".MV06.Risposta_opening,
                           Risposta_Closing => "Motors".MV06.Risposta_closing,
                           Limit_Switch_Open_HMI => "Motors".MV06.Limit_switch_open,
                           Limit_Switch_Close_HMI => "Motors".MV06.Limit_switch_close,
                           Comulativo_allarmi => "Motors".MV06.Comulativo_allarmi);
END_REGION

REGION Network 11: MV05
   RUNG wire#powerrail
      "HMI Standard Motorized Valve"(Ingresso_run_Opening := "Inputs"."MV05 RUN_Opening", Ingresso_run_Closing := "Inputs"."MV05 RUN_Closing", Allarme1 := "Allarm".MV_05_FAULT, Allarme2 := FALSE, Allarme3 := false, Allarme4 := false, Allarme5 := false, Limit_switch_Open := "Inputs"."MV05 open", Limiti_Switch_Close := "Inputs"."MV05 Close", Risposta_Opening => "Motors".MV05.Risposta_opening, Risposta_Closing => "Motors".MV05.Risposta_closing, Limit_Switch_Open_HMI => "Motors".MV05.Limit_switch_open, Limit_Switch_Close_HMI => "Motors".MV05.Limit_switch_close, Comulativo_allarmi => "Motors".MV05.Comulativo_allarmi)
   END_RUNG
   // the same network as SCL:
   "HMI Standard Motorized Valve"(Ingresso_run_Opening := "Inputs"."MV05 RUN_Opening",
                           Ingresso_run_Closing := "Inputs"."MV05 RUN_Closing",
                           Allarme1 := "Allarm".MV_05_FAULT,
                           Allarme2 := FALSE,
                           Allarme3 := false,
                           Allarme4 := false,
                           Allarme5 := false,
                           Limit_switch_Open := "Inputs"."MV05 open",
                           Limiti_Switch_Close := "Inputs"."MV05 Close",
                           Risposta_Opening => "Motors".MV05.Risposta_opening,
                           Risposta_Closing => "Motors".MV05.Risposta_closing,
                           Limit_Switch_Open_HMI => "Motors".MV05.Limit_switch_open,
                           Limit_Switch_Close_HMI => "Motors".MV05.Limit_switch_close,
                           Comulativo_allarmi => "Motors".MV05.Comulativo_allarmi);
END_REGION

REGION Network 12: MV02
   RUNG wire#powerrail
      "HMI Standard Motorized Valve"(Ingresso_run_Opening := "Inputs"."MV02 RUN_Opening", Ingresso_run_Closing := "Inputs"."MV02 RUN_Closing", Allarme1 := "Allarm".MV02_FAULT, Allarme2 := FALSE, Allarme3 := false, Allarme4 := false, Allarme5 := false, Limit_switch_Open := "Inputs"."MV02 Open", Limiti_Switch_Close := "Inputs"."MV02 Close", Risposta_Opening => "Motors".MV02.Risposta_opening, Risposta_Closing => "Motors".MV02.Risposta_closing, Limit_Switch_Open_HMI => "Motors".MV02.Limit_switch_open, Limit_Switch_Close_HMI => "Motors".MV02.Limit_switch_close, Comulativo_allarmi => "Motors".MV02.Comulativo_allarmi)
   END_RUNG
   // the same network as SCL:
   "HMI Standard Motorized Valve"(Ingresso_run_Opening := "Inputs"."MV02 RUN_Opening",
                           Ingresso_run_Closing := "Inputs"."MV02 RUN_Closing",
                           Allarme1 := "Allarm".MV02_FAULT,
                           Allarme2 := FALSE,
                           Allarme3 := false,
                           Allarme4 := false,
                           Allarme5 := false,
                           Limit_switch_Open := "Inputs"."MV02 Open",
                           Limiti_Switch_Close := "Inputs"."MV02 Close",
                           Risposta_Opening => "Motors".MV02.Risposta_opening,
                           Risposta_Closing => "Motors".MV02.Risposta_closing,
                           Limit_Switch_Open_HMI => "Motors".MV02.Limit_switch_open,
                           Limit_Switch_Close_HMI => "Motors".MV02.Limit_switch_close,
                           Comulativo_allarmi => "Motors".MV02.Comulativo_allarmi);
END_REGION

REGION Network 13: MV01
